// TwinCAT 3 PLC project CandyVendingMachine
// ProgramVersion: 3.1.4026.11
// libraries:
//   Tc2_Standard, * (Beckhoff Automation GmbH)
//   Tc2_System, * (Beckhoff Automation GmbH)
//   Tc2_Utilities, * (Beckhoff Automation GmbH)
// project tree:
//   AnyToArg/Classes/ AnyToTArgConverter.TcPOU
//   Candies/Classes/ AbstractCandy.TcPOU, Alpenliebe.TcPOU, Altoids.TcPOU, BobsSweetStripes.TcPOU, BrachsCandyCorn.TcPOU, ChupaChups.TcPOU, Goldbears.TcPOU, MnMs.TcPOU, Poppins.TcPOU, SkittlesSour.TcPOU, SnickersBar.TcPOU, TwizzlersLicorizeTwists.TcPOU, WonkaGobstopper.TcPOU
//   Candies/Types/Aliases/ CandyAmountInGram.TcDUT, CandyName.TcDUT
//   Candies/Types/Enums/ CandyTypes.TcDUT
//   CandyConsumer/Classes/ AbstractCandyConsumer.TcPOU
//   CandyConsumer/Types/Aliases/ ConsumerName.TcDUT, SatisfactionLevelInPercent.TcDUT
//   CandyDispatchers/Classes/ AbstractCandyDispatcher.TcPOU, CandyBarDispatcher.TcPOU, CandyCornDispatcher.TcPOU, CandyDispatcherFactory.TcPOU, CandySticksDispatcher.TcPOU, CaramelCandyDispatcher.TcPOU, ChoclateCandyDispatcher.TcPOU, GummyCandyDispatcher.TcPOU, HardCandyDispatcher.TcPOU, JawbreakersDispatcher.TcPOU, LicoriceCandyDispatcher.TcPOU, LollipopsDispatcher.TcPOU, MintsDispatcher.TcPOU, SourCandyDispatcher.TcPOU
//   CandyMachineProvider/Classes/ CandyMachineProvider.TcPOU, NinjaIncCandyMachineProvider.TcPOU
//   CandyMachine/Classes/ AbstractCandyMachine.TcPOU, CommonCandyMachine.TcPOU, GreedyCandyMachine.TcPOU, PickyCandyMachine.TcPOU
//   Logger/Classes/ AbstractLogger.TcPOU (not stored), AdsLogger.TcPOU, AdsLogMessage.TcPOU, LoggerProvider.TcPOU
//   NinjaCandyBehavior/Classes/ AbstractNinjaCandyConsumeBehavior.TcPOU, CommonNinjaCandyBehavior.TcPOU, GreedyNinjaCandyBehavior.TcPOU, PickyNinjaCandyBehavior.TcPOU
//   NinjaCandyBehavior/types/Enums/ ConsumerTypes.TcDUT, TasteScale.TcDUT
//   NinjaMonkeys/Classes/ AjninsCandyPreferences.TcPOU, IndividualCandyPreferences.TcPOU, NinjaMonkey.TcPOU
//   Tasks/Main/ MAIN.TcPOU, PlcTask.TcTTO
// real-time tasks:
//   TASK PlcTask: cycle T#10ms, priority 20, ADS port 350

CONFIGURATION CandyVendingMachine
    RESOURCE PLC ON TwinCAT3
        TASK PlcTask(INTERVAL := T#10ms, PRIORITY := 20);
        PROGRAM MAIN WITH PlcTask : MAIN;
    END_RESOURCE
END_CONFIGURATION

// ---- Candies/Types/Aliases/CandyAmountInGram.TcDUT
(*

short summary
=============
Alias of the subrange UINT(0..500).
It's used for the candy amount. The candy
machine is able to handle packaging units up
to 500 grams

legal notes
===========
SPDX-FileCopyrightText: © 2024 ekvip automation GmbH <info@ekvip.de>
SPDX-License-Identifier: Apache-2.0
For details check: Apache-2.0_

.. _Apache-2.0: https://www.apache.org/licenses/LICENSE-2.0

*)

TYPE CandyAmountInGram : 
	UINT(0..500); 
END_TYPE

// ---- Candies/Types/Aliases/CandyName.TcDUT
(*

short summary
=============
T_MaxString alias for the candy name.  

legal notes
===========
SPDX-FileCopyrightText: © 2024 ekvip automation GmbH <info@ekvip.de>
SPDX-License-Identifier: Apache-2.0
For details check: Apache-2.0_

.. _Apache-2.0: https://www.apache.org/licenses/LICENSE-2.0

*)

TYPE CandyName :
	Tc2_System.T_MaxString; 
END_TYPE

// ---- Candies/Types/Enums/CandyTypes.TcDUT
(*

short summary
=============
Enumeration of the candy types.
A single bit represents each candy type.
The candy type is stored in a word => so there can be
16 different candy types.
As a sweet usually consists of a mixture of different types, 
the enumeration is not strict. 
Each sweet can save its type by setting the corresponding bits. 

legal notes
===========
SPDX-FileCopyrightText: © 2024 ekvip automation GmbH <info@ekvip.de>
SPDX-License-Identifier: Apache-2.0
For details check: Apache-2.0_

.. _Apache-2.0: https://www.apache.org/licenses/LICENSE-2.0

*)

{attribute 'qualified_only'}
{attribute 'to_string'}
TYPE CandyTypes :
(
	(* bit 0 is type candy bar like a snickers *)
	CANDY_BARS		:= 16#0001,
	(* bit 1 is type candy corn like brach's candy corn *)
	CANDY_CORN		:= 16#0002,
	(* bit 2 is type stick candy like a christmas candy cane *)
	CANDY_STICKS	:= 16#0004,
	(* bit 3 is type caramel candy like omar cream *)
	CARAMEL_CANDY	:= 16#0008,
	(* bit 4 is type choclate candy like hershey *)
	CHOCOLATE_CANDY	:= 16#0010,
	(* bit 5 is type gummie candy like haribo *)
	GUMMY_CANDY		:= 16#0020,
	(* bit 6 is type mints like altoids *)
	MINTS			:= 16#0040,
	(* bit 7 is type lollipop like chupa chups *)
	LOLLIPOPS		:= 16#0080,
	(* bit 8 is type jawbreakers like willy wonka's everlasting gobstopper *) 
	JAWBREAKERS		:= 16#0100,
	(* bit 9 is type hard candy like pass pass pulse *)
	HARD_CANDY		:= 16#0200,
	(* bit 10 is type licorice candy like lakrids bülow *)
	LICORICE_CANDY	:= 16#0400,
	(* bit 11 is type sour candy like warheads *)
	SOUR_CANDY		:= 16#0800 	
)WORD;
END_TYPE

// ---- CandyConsumer/Types/Aliases/ConsumerName.TcDUT
(*

short summary
=============
A T_MaxString alias for the consumer name

legal notes
===========
SPDX-FileCopyrightText: © 2024 ekvip automation GmbH <info@ekvip.de>
SPDX-License-Identifier: Apache-2.0
For details check: Apache-2.0_

.. _Apache-2.0: https://www.apache.org/licenses/LICENSE-2.0

*)

TYPE ConsumerName :
	Tc2_System.T_MaxString; 
END_TYPE

// ---- CandyConsumer/Types/Aliases/SatisfactionLevelInPercent.TcDUT
(*

short summary
=============
alias for an unit subrange form 0 to 100.
It is used as satisfaction level for the candy consumer.
0 means depression
100 means euphoria

legal notes
===========
SPDX-FileCopyrightText: © 2024 ekvip automation GmbH <info@ekvip.de>
SPDX-License-Identifier: Apache-2.0
For details check: Apache-2.0_

.. _Apache-2.0: https://www.apache.org/licenses/LICENSE-2.0

*)

TYPE SatisfactionLevelInPercent :
	UINT(0..100); 
END_TYPE

// ---- NinjaCandyBehavior/types/Enums/ConsumerTypes.TcDUT
(*

short summary
=============
The world is full of different consumer types
but we've only defined two of it.
The greedy consumer (more is better)
The picky consumer (it's only worth it if it's good)

legal notes
===========
SPDX-FileCopyrightText: © 2024 ekvip automation GmbH <info@ekvip.de>
SPDX-License-Identifier: Apache-2.0
For details check: Apache-2.0_

.. _Apache-2.0: https://www.apache.org/licenses/LICENSE-2.0

*)

{attribute 'qualified_only'}
{attribute 'strict'}
{attribute 'to_string'}
TYPE ConsumerTypes :
(
	(* common neither picky nor greedy *)
	COMMON := 0,
	(* cookie monster style *)
	GREEDY,
	(* finicky style *)
	PICKY
)UDINT;
END_TYPE

// ---- NinjaCandyBehavior/types/Enums/TasteScale.TcDUT
(*

short summary
=============
This is enumeration is used as factor
to calculate the satisfaction level of the consumer.

legal notes
===========
SPDX-FileCopyrightText: © 2024 ekvip automation GmbH <info@ekvip.de>
SPDX-License-Identifier: Apache-2.0
For details check: Apache-2.0_

.. _Apache-2.0: https://www.apache.org/licenses/LICENSE-2.0

*)

{attribute 'qualified_only'}
{attribute 'strict'}
{attribute 'to_string'}
TYPE TasteScale :
(
	(* decreases maybe consumers statisfaction level *)
	DISGUSTING := -1,
	(* has maybe no effect on the consumers statisfaction level *)
	OKAY := 0,
	(* increases maybe consumers statisfaction level *)
	DELICIOUS := 1
)DINT := OKAY;
END_TYPE

// ---- Tasks/Main/MAIN.TcPOU
(*

short summary
=============
this is the main task of the
candy vending machine application

legal notes
===========
SPDX-FileCopyrightText: © 2024 ekvip automation GmbH <info@ekvip.de>
SPDX-License-Identifier: Apache-2.0
For details check: Apache-2.0_

.. _Apache-2.0: https://www.apache.org/licenses/LICENSE-2.0

*)

PROGRAM MAIN
VAR
	(* to print the log messages with the run method of the logger *)
	loggingProvider :LoggerProvider(0);
	(* behavior for a greedy candy consuming ninja *)
	greedy				:GreedyNinjaCandyBehavior(0);
	(* behavior for a picky candy consuming ninja *)
	picky				:PickyNinjaCandyBehavior(0);
	(* candy preferences of Ajnin *)
	ajninPreferences	:AjninsCandyPreferences();
	(* yeknom as candy consumer *)
	yeknom				:NinjaMonkey(greedy,0);
	(* ajnin as candy consumer *)
	ajnin				:NinjaMonkey(picky, ajninPreferences);
	(* rising edge will feed Ajnin *)
	feedAjnin			:BOOL;
	(* rising edge will feed Yeknom *)
	feedYeknom			:BOOL; 
END_VAR

ajnin.lootCandies(feedAjnin);
yeknom.lootCandies(feedYeknom);
loggingProvider.logger.run();

END_PROGRAM

// ---- Logger/Classes/LoggerProvider.TcPOU
(*

short summary
=============
A layer to hide the concrete used logger
and to make it easy to use the same logger

legal notes
===========
SPDX-FileCopyrightText: © 2024 ekvip automation GmbH <info@ekvip.de>
SPDX-License-Identifier: Apache-2.0
For details check: Apache-2.0_

.. _Apache-2.0: https://www.apache.org/licenses/LICENSE-2.0

*)

FUNCTION_BLOCK LoggerProvider
VAR_STAT
	(* differnt logger injected from outside *)
	injectedLogger	:REFERENCE TO AbstractLogger;
	(* default logger if nothing was injected *)
	defaultLogger 	:AdsLogger();
END_VAR

(*

short summary
=============
this method provides the possibility
to use a differnt logger for example
a file logger. 

legal notes
===========
SPDX-FileCopyrightText: © 2024 ekvip automation GmbH <info@ekvip.de>
SPDX-License-Identifier: Apache-2.0
For details check: Apache-2.0_

.. _Apache-2.0: https://www.apache.org/licenses/LICENSE-2.0

*)

METHOD FB_init :BOOL
VAR_INPUT
	(* if TRUE, the retain variables are initialized (warm start / cold start) *)
	bInitRetains	:BOOL;
	(* if TRUE, the instance afterwards gets moved into the copy code (online change) *) 
	bInCopyCode		:BOOL;
	(* if no other logger is required then use just 0 as parameter *)
	otherLogger		:REFERENCE TO AbstractLogger;
END_VAR
IF (__ISVALIDREF(otherLogger) AND_THEN NOT __ISVALIDREF(THIS^.injectedLogger)) THEN
	THIS^.injectedLogger REF= otherLogger;
END_IF
END_METHOD

(*

short summary
=============
property to get the used logger instance
 
legal notes
===========
SPDX-FileCopyrightText: © 2024 ekvip automation GmbH <info@ekvip.de>
SPDX-License-Identifier: Apache-2.0
For details check: Apache-2.0_

.. _Apache-2.0: https://www.apache.org/licenses/LICENSE-2.0

*)

PROPERTY logger :REFERENCE TO AbstractLogger
GET
(*

short summary
=============
getter of the property to get the used logger instance

legal notes
===========
SPDX-FileCopyrightText: © 2024 ekvip automation GmbH <info@ekvip.de>
SPDX-License-Identifier: Apache-2.0
For details check: Apache-2.0_

.. _Apache-2.0: https://www.apache.org/licenses/LICENSE-2.0

*)

VAR
END_VAR
IF (__ISVALIDREF(THIS^.injectedLogger)) THEN
	logger REF= THIS^.injectedLogger;
ELSE
	logger REF= THIS^.defaultLogger;
END_IF
END_GET
END_PROPERTY

END_FUNCTION_BLOCK

// ---- Logger/Classes/AdsLogger.TcPOU
(*

short summary
=============
a logger to write ADSLOG messages 

legal notes
===========
SPDX-FileCopyrightText: © 2024 ekvip automation GmbH <info@ekvip.de>
SPDX-License-Identifier: Apache-2.0
For details check: Apache-2.0_

.. _Apache-2.0: https://www.apache.org/licenses/LICENSE-2.0

*)

FUNCTION_BLOCK AdsLogger EXTENDS AbstractLogger
VAR
	(* buffer to store the messages *)
	messages		:POINTER TO POINTER TO AdsLogMessage;
	(* size of the message buffer *)
	size			:DWORD;
	(* the message buffer is a simple ring buffer this the read pointer for it *)
	readPointer		:DWORD := 0;
	(* the message buffer is a simple ring buffer this the write pointer for it *)
	writePointer	:DWORD := 0;
END_VAR
VAR CONSTANT
	(* inital message buffer size *) 
	MIN_BUFFER_SIZE :DWORD := 255;
END_VAR

(*

short summary
=============
this method appends a log message to the message buffer

legal notes
===========
SPDX-FileCopyrightText: © 2024 ekvip automation GmbH <info@ekvip.de>
SPDX-License-Identifier: Apache-2.0
For details check: Apache-2.0_

.. _Apache-2.0: https://www.apache.org/licenses/LICENSE-2.0

*)

METHOD PRIVATE appendNewMessage
VAR_INPUT
	(* ADSLOG message mask *)
	messageType :DWORD;
END_VAR
VAR_IN_OUT
	(* content of the log message *)
	message :Tc2_System.T_MaxString;
END_VAR
VAR
	(* pointer to the new log message *) 
	new	:POINTER TO AdsLogMessage;
END_VAR
IF (THIS^.isBufferFull OR (THIS^.messages = 0)) THEN
	THIS^.resize();
END_IF
RETURN((THIS^.messages = 0) OR_ELSE THIS^.isBufferFull);

new := __NEW(AdsLogMessage(msg := message, msgType := messageType));
RETURN(new = 0);
THIS^.messages[THIS^.writePointer] := new;
THIS^.writePointer := THIS^.incrementBufferPointer(THIS^.writePointer);
END_METHOD

(*

short summary
=============
writes a log message for a critical event
It will be stored in the twinCAT logbook 
and open a message box

legal notes
===========
SPDX-FileCopyrightText: © 2024 ekvip automation GmbH <info@ekvip.de>
SPDX-License-Identifier: Apache-2.0
For details check: Apache-2.0_

.. _Apache-2.0: https://www.apache.org/licenses/LICENSE-2.0

*)

METHOD critical
VAR_INPUT
	(* log message to write *)
	message :Tc2_System.T_MaxString;
END_VAR
THIS^.appendNewMessage(
	Tc2_System.ADSLOG_MSGTYPE_ERROR OR Tc2_System.ADSLOG_MSGTYPE_RESOURCE OR Tc2_System.ADSLOG_MSGTYPE_MSGBOX, 
	message
);
END_METHOD

(*

short summary
=============
method to log a debug message

legal notes
===========
SPDX-FileCopyrightText: © 2024 ekvip automation GmbH <info@ekvip.de>
SPDX-License-Identifier: Apache-2.0
For details check: Apache-2.0_

.. _Apache-2.0: https://www.apache.org/licenses/LICENSE-2.0

*)

METHOD debug
VAR_INPUT
	(* log message to write *)
	message :Tc2_System.T_MaxString;
END_VAR
THIS^.appendNewMessage(Tc2_System.ADSLOG_MSGTYPE_HINT, message);
END_METHOD

(*

short summary
=============
method to log a error message

legal notes
===========
SPDX-FileCopyrightText: © 2024 ekvip automation GmbH <info@ekvip.de>
SPDX-License-Identifier: Apache-2.0
For details check: Apache-2.0_

.. _Apache-2.0: https://www.apache.org/licenses/LICENSE-2.0

*)

METHOD error
VAR_INPUT
	(* log message to write *)
	message :Tc2_System.T_MaxString;
END_VAR
THIS^.appendNewMessage(Tc2_System.ADSLOG_MSGTYPE_ERROR, message);
END_METHOD

(*

short summary
=============
this method clean up the memory
(free it again)

legal notes
===========
SPDX-FileCopyrightText: © 2024 ekvip automation GmbH <info@ekvip.de>
SPDX-License-Identifier: Apache-2.0
For details check: Apache-2.0_

.. _Apache-2.0: https://www.apache.org/licenses/LICENSE-2.0

*)

METHOD FB_exit :BOOL
VAR_INPUT
	(* if TRUE, the exit method is called for exiting an instance that is copied afterwards (online change). *)
	bInCopyCode :BOOL;
END_VAR
VAR
	(* buffer pointer to free the message buffer memory again *)
	buffer 		:POINTER TO __XWORD;
END_VAR
RETURN(THIS^.messages = 0);
WHILE (NOT THIS^.isBufferEmpty) DO
	THIS^.printMessage();
END_WHILE
buffer := THIS^.messages;
__DELETE(buffer);
THIS^.messages := 0;
THIS^.size := 0;
THIS^.writePointer := 0;
THIS^.readPointer := 0;
END_METHOD

(*

short summary
=============
method to increment the read and write pointer
of the message buffer

legal notes
===========
SPDX-FileCopyrightText: © 2024 ekvip automation GmbH <info@ekvip.de>
SPDX-License-Identifier: Apache-2.0
For details check: Apache-2.0_

.. _Apache-2.0: https://www.apache.org/licenses/LICENSE-2.0

*)

METHOD PRIVATE incrementBufferPointer :DWORD
VAR_INPUT
	(* current pointer value *)
	bufferPointer :DWORD;
END_VAR
incrementBufferPointer := ((bufferPointer + 1) MOD THIS^.size);
END_METHOD

(*

short summary
=============
method to log a info message

legal notes
===========
SPDX-FileCopyrightText: © 2024 ekvip automation GmbH <info@ekvip.de>
SPDX-License-Identifier: Apache-2.0
For details check: Apache-2.0_

.. _Apache-2.0: https://www.apache.org/licenses/LICENSE-2.0

*)

METHOD info
VAR_INPUT
	(* log message to write *)
	message :Tc2_System.T_MaxString;
END_VAR
THIS^.appendNewMessage(Tc2_System.ADSLOG_MSGTYPE_HINT, message);
END_METHOD

(*

short summary
=============
property to check if the
ring buffer is empty

legal notes
===========
SPDX-FileCopyrightText: © 2024 ekvip automation GmbH <info@ekvip.de>
SPDX-License-Identifier: Apache-2.0
For details check: Apache-2.0_

.. _Apache-2.0: https://www.apache.org/licenses/LICENSE-2.0

*)

PROPERTY PRIVATE isBufferEmpty :BOOL
GET
(*

short summary
=============
getter of the property to check if the
ring buffer is empty

legal notes
===========
SPDX-FileCopyrightText: © 2024 ekvip automation GmbH <info@ekvip.de>
SPDX-License-Identifier: Apache-2.0
For details check: Apache-2.0_

.. _Apache-2.0: https://www.apache.org/licenses/LICENSE-2.0

*)

VAR
END_VAR
isBufferEmpty := (THIS^.readPointer = THIS^.writePointer);
END_GET
END_PROPERTY

(*

short summary
=============
property to check if the
ring buffer is full

legal notes
===========
SPDX-FileCopyrightText: © 2024 ekvip automation GmbH <info@ekvip.de>
SPDX-License-Identifier: Apache-2.0
For details check: Apache-2.0_

.. _Apache-2.0: https://www.apache.org/licenses/LICENSE-2.0

*)

PROPERTY PRIVATE isBufferFull :BOOL
GET
(*

short summary
=============
getter of the property to check if the
ring buffer is full

legal notes
===========
SPDX-FileCopyrightText: © 2024 ekvip automation GmbH <info@ekvip.de>
SPDX-License-Identifier: Apache-2.0
For details check: Apache-2.0_

.. _Apache-2.0: https://www.apache.org/licenses/LICENSE-2.0

*)

VAR
END_VAR
isBufferFull := (THIS^.incrementBufferPointer(THIS^.writePointer) = THIS^.readPointer);
END_GET
END_PROPERTY

(*

short summary
=============
method to write the log message to
ADSLOG and it frees the memory of
the message again

legal notes
===========
SPDX-FileCopyrightText: © 2024 ekvip automation GmbH <info@ekvip.de>
SPDX-License-Identifier: Apache-2.0
For details check: Apache-2.0_

.. _Apache-2.0: https://www.apache.org/licenses/LICENSE-2.0

*)

METHOD PRIVATE printMessage
VAR
	(* message pointer to free the memory again *)
	msg :POINTER TO AdsLogMessage;
END_VAR
IF (THIS^.messages[THIS^.readPointer] <> 0) THEN
	Tc2_System.ADSLOGSTR(
		msgCtrlMask := THIS^.messages[THIS^.readPointer]^.messageType,
		msgFmtStr := '%s',
		strArg := THIS^.messages[THIS^.readPointer]^.message
	);
	msg := THIS^.messages[THIS^.readPointer];
	__DELETE(msg);
	THIS^.messages[THIS^.readPointer] := 0;
END_IF
THIS^.readPointer := THIS^.incrementBufferPointer(THIS^.readPointer);
END_METHOD

(*

short summary
=============
this method resizes the messages buffer
if it is full or not created

legal notes
===========
SPDX-FileCopyrightText: © 2024 ekvip automation GmbH <info@ekvip.de>
SPDX-License-Identifier: Apache-2.0
For details check: Apache-2.0_

.. _Apache-2.0: https://www.apache.org/licenses/LICENSE-2.0

*)

METHOD PRIVATE resize
VAR
	(* new buffer for the messages array *)
	newBuffer 			:POINTER TO __XWORD;
	(* just to free the memory again *)
	oldBuffer 			:POINTER TO __XWORD;
	(* pointer with the smaller value *)
	minPointer  		:DWORD;
	(* pointer with the bigger value *)
	maxPointer  		:DWORD;
	(* new position in new message buffer of the pointer with the bigger value *)
	newMaxPointerPos	:DWORD;
	(* number of elements to copy for the pointer with the bigger value *)
	amountMaxPointer	:DWORD;
	(* new size of the messages buffer *)
	newSize 			:DWORD;
END_VAR
newSize := MAX(THIS^.MIN_BUFFER_SIZE, THIS^.size * 2);
RETURN(newSize < THIS^.size);
newBuffer := __NEW(__XWORD, newSize);
RETURN(newBuffer = 0);
IF (NOT THIS^.isBufferEmpty) THEN
	minPointer := MIN(THIS^.writePointer, THIS^.readPointer);
	maxPointer := MAX(THIS^.writePointer, THIS^.readPointer);
	amountMaxPointer := SEL(
		((THIS^.size-1) = maxPointer),
		((THIS^.size-1)-maxPointer),
		THIS^.size-1
	);
	newMaxPointerPos := ((newSize-1)-amountMaxPointer);
	Tc2_System.MEMCPY(
		destAddr	:= newBuffer,
		srcAddr		:= THIS^.messages,
		n			:= ((minPointer+1)*SIZEOF(__XWORD))
	);
	Tc2_System.MEMCPY(
		destAddr	:= ADR(newBuffer[SEL(((THIS^.size-1) = maxPointer),newMaxPointerPos,minPointer+1)]),
		srcAddr		:= ADR(THIS^.messages[minPointer+1]),
		n			:= (amountMaxPointer*SIZEOF(__XWORD))
	);
	IF (THIS^.readPointer > THIS^.writePointer) THEN
		THIS^.readPointer := newMaxPointerPos;
	ELSE
		THIS^.writePointer := newMaxPointerPos;
	END_IF
END_IF
IF (THIS^.messages <> 0) THEN
	oldBuffer := THIS^.messages;
	__DELETE(oldBuffer);
END_IF
THIS^.messages := newBuffer;
THIS^.size := newSize;
END_METHOD

(*

short summary
=============
fetches the messages from buffer and
writes it to ADSLOG. This method must
be called cyclic.

legal notes
===========
SPDX-FileCopyrightText: © 2024 ekvip automation GmbH <info@ekvip.de>
SPDX-License-Identifier: Apache-2.0
For details check: Apache-2.0_

.. _Apache-2.0: https://www.apache.org/licenses/LICENSE-2.0

*)

METHOD run
VAR_INST
	(* TON timer to write the messages in a serial way *)
	printNextMsg	:Tc2_Standard.TON;	
END_VAR
RETURN(THIS^.messages = 0);
printNextMsg(IN:= TRUE, PT:=T#30MS);
RETURN(NOT printNextMsg.Q);
RETURN(THIS^.isBufferEmpty);
printNextMsg(IN:= FALSE);
THIS^.printMessage();
END_METHOD

(*

short summary
=============
method to log a warning message

legal notes
===========
SPDX-FileCopyrightText: © 2024 ekvip automation GmbH <info@ekvip.de>
SPDX-License-Identifier: Apache-2.0
For details check: Apache-2.0_

.. _Apache-2.0: https://www.apache.org/licenses/LICENSE-2.0

*)

METHOD warning
VAR_INPUT
	(* log message to write *)
	message :Tc2_System.T_MaxString;
END_VAR
THIS^.appendNewMessage(Tc2_System.ADSLOG_MSGTYPE_WARN, message);
END_METHOD

END_FUNCTION_BLOCK

// ---- Logger/Classes/AdsLogMessage.TcPOU
(*

short summary
=============
just a dto to store the logging data for
the ads logger

legal notes
===========
SPDX-FileCopyrightText: © 2024 ekvip automation GmbH <info@ekvip.de>
SPDX-License-Identifier: Apache-2.0
For details check: Apache-2.0_

.. _Apache-2.0: https://www.apache.org/licenses/LICENSE-2.0

*)

{attribute 'enable_dynamic_creation'}
FUNCTION_BLOCK AdsLogMessage
VAR
	(* log message content *)
	msg		:Tc2_System.T_MaxString;
	(* ADSLOG message type mask *)
	msgType	:DWORD;
END_VAR

(*

short summary
=============
initialize the message values

legal notes
===========
SPDX-FileCopyrightText: © 2024 ekvip automation GmbH <info@ekvip.de>
SPDX-License-Identifier: Apache-2.0
For details check: Apache-2.0_

.. _Apache-2.0: https://www.apache.org/licenses/LICENSE-2.0

*)

METHOD FB_init :BOOL
VAR_INPUT
	(* if TRUE, the retain variables are initialized (warm start / cold start) *)
	bInitRetains	:BOOL;
	(* if TRUE, the instance afterwards gets moved into the copy code (online change) *) 
	bInCopyCode		:BOOL;
	(* content of the message *)
	msg				:Tc2_System.T_MaxString;
	(* mask of an ADSLOG *)
	msgType			:DWORD;
END_VAR
THIS^.msg := msg;
THIS^.msgType := msgType;
END_METHOD

(*

short summary
=============
property to get the message content

legal notes
===========
SPDX-FileCopyrightText: © 2024 ekvip automation GmbH <info@ekvip.de>
SPDX-License-Identifier: Apache-2.0
For details check: Apache-2.0_

.. _Apache-2.0: https://www.apache.org/licenses/LICENSE-2.0

*)

PROPERTY message :Tc2_System.T_MaxString
GET
(*

short summary
=============
getter of the property to get the message content

legal notes
===========
SPDX-FileCopyrightText: © 2024 ekvip automation GmbH <info@ekvip.de>
SPDX-License-Identifier: Apache-2.0
For details check: Apache-2.0_

.. _Apache-2.0: https://www.apache.org/licenses/LICENSE-2.0

*)

VAR
END_VAR
message := THIS^.msg;
END_GET
END_PROPERTY

(*

short summary
=============
property to get the ads message type mask

legal notes
===========
SPDX-FileCopyrightText: © 2024 ekvip automation GmbH <info@ekvip.de>
SPDX-License-Identifier: Apache-2.0
For details check: Apache-2.0_

.. _Apache-2.0: https://www.apache.org/licenses/LICENSE-2.0

*)

PROPERTY messageType :DWORD
GET
(*

short summary
=============
getter of the property to get the ads message type mask

legal notes
===========
SPDX-FileCopyrightText: © 2024 ekvip automation GmbH <info@ekvip.de>
SPDX-License-Identifier: Apache-2.0
For details check: Apache-2.0_

.. _Apache-2.0: https://www.apache.org/licenses/LICENSE-2.0

*)

VAR
END_VAR
messageType := THIS^.msgType;
END_GET
END_PROPERTY

END_FUNCTION_BLOCK

// ---- NinjaCandyBehavior/Classes/GreedyNinjaCandyBehavior.TcPOU
(*

short summary
=============
the behavior of a greedy ninja

legal notes
===========
SPDX-FileCopyrightText: © 2024 ekvip automation GmbH <info@ekvip.de>
SPDX-License-Identifier: Apache-2.0
For details check: Apache-2.0_

.. _Apache-2.0: https://www.apache.org/licenses/LICENSE-2.0

*)

FUNCTION_BLOCK GreedyNinjaCandyBehavior EXTENDS AbstractNinjaCandyConsumeBehavior
VAR_STAT
	(* default provider for the greedies*)
	greedyDefaultProvider :NinjaIncCandyMachineProvider(ConsumerTypes.GREEDY);
END_VAR

(*

short summary
=============
This method calculates the satisfaction level
for a candy eating greedy consumer.

legal notes
===========
SPDX-FileCopyrightText: © 2024 ekvip automation GmbH <info@ekvip.de>
SPDX-License-Identifier: Apache-2.0
For details check: Apache-2.0_

.. _Apache-2.0: https://www.apache.org/licenses/LICENSE-2.0

*)

METHOD  calculateSatisfactionLevel
VAR_INPUT
	(* taste scale of candy *)
	tastiness				:TasteScale;
	(* amount of the candies to eat *)
	amountOfCandy			:CandyAmountInGram;
END_VAR
VAR_IN_OUT
	(* the satisfaction level of the consumer *)
	actualSatisfactionLevel	:SatisfactionLevelInPercent;
END_VAR
VAR CONSTANT
	(* maximum possible satisfaction level*)
	MAX_SATISFACTION 		:SatisfactionLevelInPercent := 100;
	(* it is a lower limit as it is named *)
	AVOID_DIVISON_BY_ZERO 	:SatisfactionLevelInPercent := 1;
	(* factor for the greediness of the consumer *)
	GREEDINESS				:SatisfactionLevelInPercent := 78;
	(* for one a candy package the maximum amount *)
	MAX_AMOUNT				:CandyAmountInGram := 500;
END_VAR
RETURN(actualSatisfactionLevel >= MAX_SATISFACTION);

{warning disable C0196}
{warning disable C0197}
actualSatisfactionLevel := TO_UINT(
	actualSatisfactionLevel + TO_SINT(
		LOG(
			TO_REAL(MAX_SATISFACTION)
			/TO_REAL(LIMIT(AVOID_DIVISON_BY_ZERO, actualSatisfactionLevel, MAX_SATISFACTION))
		) * (
			TO_REAL(amountOfCandy)
			/TO_REAL(MAX_AMOUNT)
		)
		* (MAX_SATISFACTION - GREEDINESS)
	)
);
{warning restore C0196}
{warning restore C0197}
END_METHOD

(*

short summary
=============
inject the candy vending machine provider
during declaration.

legal notes
===========
SPDX-FileCopyrightText: © 2024 ekvip automation GmbH <info@ekvip.de>
SPDX-License-Identifier: Apache-2.0
For details check: Apache-2.0_

.. _Apache-2.0: https://www.apache.org/licenses/LICENSE-2.0

*)

METHOD FB_init :BOOL
VAR_INPUT
	(* if TRUE, the retain variables are initialized (warm start / cold start) *)
	bInitRetains		:BOOL;
	(* if TRUE, the instance afterwards gets moved into the copy code (online change) *)
	bInCopyCode			:BOOL;
	(* candy vending machine provider for the consumer *)
	candyMachineProvider:REFERENCE TO CandyMachineProvider;
END_VAR
IF (__ISVALIDREF(candyMachineProvider)) THEN
	THIS^.candyMachineProvider REF= candyMachineProvider;
ELSE
	THIS^.candyMachineProvider REF= THIS^.greedyDefaultProvider;
END_IF
END_METHOD

END_FUNCTION_BLOCK

// ---- NinjaCandyBehavior/Classes/AbstractNinjaCandyConsumeBehavior.TcPOU
(*

short summary
=============
different consumers have a different
behavior. This class is to decouple
behavior from the consumer.

legal notes
===========
SPDX-FileCopyrightText: © 2024 ekvip automation GmbH <info@ekvip.de>
SPDX-License-Identifier: Apache-2.0
For details check: Apache-2.0_

.. _Apache-2.0: https://www.apache.org/licenses/LICENSE-2.0

*)

FUNCTION_BLOCK ABSTRACT AbstractNinjaCandyConsumeBehavior
VAR
	(* candy vending machine provider to get a machine to loot *)
	candyMachineProvider	:REFERENCE TO CandyMachineProvider;
END_VAR
VAR_STAT
	(* default provider *)
	defaultProvider :NinjaIncCandyMachineProvider(ConsumerTypes.COMMON);
END_VAR

(*

short summary
=============
This method calculates the satisfaction level if the consumer
eates some candies.

legal notes
===========
SPDX-FileCopyrightText: © 2024 ekvip automation GmbH <info@ekvip.de>
SPDX-License-Identifier: Apache-2.0
For details check: Apache-2.0_

.. _Apache-2.0: https://www.apache.org/licenses/LICENSE-2.0

*)

METHOD ABSTRACT calculateSatisfactionLevel
VAR_INPUT
	(* taste scale of candy *)
	tastiness				:TasteScale;
	(* amount of the candies to eat *)
	amountOfCandy			:CandyAmountInGram;
END_VAR
VAR_IN_OUT
	(* the satisfaction level of the consumer *)
	actualSatisfactionLevel	:SatisfactionLevelInPercent;
END_VAR
END_METHOD

(*

short summary
=============
inject the candy vending machine provider
during declaration.

legal notes
===========
SPDX-FileCopyrightText: © 2024 ekvip automation GmbH <info@ekvip.de>
SPDX-License-Identifier: Apache-2.0
For details check: Apache-2.0_

.. _Apache-2.0: https://www.apache.org/licenses/LICENSE-2.0

*)

METHOD FB_init :BOOL
VAR_INPUT
	(* if TRUE, the retain variables are initialized (warm start / cold start) *)
	bInitRetains		:BOOL;
	(* if TRUE, the instance afterwards gets moved into the copy code (online change) *)
	bInCopyCode			:BOOL;
	(* candy vending machine provider for the consumer *)
	candyMachineProvider:REFERENCE TO CandyMachineProvider;
END_VAR
IF (__ISVALIDREF(candyMachineProvider)) THEN
	THIS^.candyMachineProvider REF= candyMachineProvider;
ELSE
	THIS^.candyMachineProvider REF= THIS^.defaultProvider;
END_IF
END_METHOD

(*

short summary
=============
this method is for the looting behavior
of the picky consumer. 
The picky consumer tries to by delcious candy only.

legal notes
===========
SPDX-FileCopyrightText: © 2024 ekvip automation GmbH <info@ekvip.de>
SPDX-License-Identifier: Apache-2.0
For details check: Apache-2.0_

.. _Apache-2.0: https://www.apache.org/licenses/LICENSE-2.0

*)

METHOD  lootACandyMachine
VAR_INPUT
	(* consumer who loots a candy vending machine *)
	consumer :REFERENCE TO AbstractCandyConsumer;
	(* preferences of consumer no preference means consumer likes every candy *)
	preferences	:REFERENCE TO IndividualCandyPreferences REF= 0;
END_VAR
VAR
	(* for-loop counter *)
	candyToEat		:CandyTypes;
	(* used candy vending machine *)
	candyMachine	:REFERENCE TO AbstractCandyMachine;
	(* the candy to eat *)
	candy			:REFERENCE TO AbstractCandy;
END_VAR
RETURN(NOT __ISVALIDREF(consumer));
candyMachine REF= THIS^.candyMachineProvider.getACandyMachine();
RETURN(NOT __ISVALIDREF(candyMachine));

FOR candyToEat := CandyTypes.CANDY_BARS TO CandyTypes.SOUR_CANDY BY candyToEat DO
	IF (__ISVALIDREF(preferences) AND_THEN preferences.howIsTheCandy(candyToEat) <> TasteScale.DELICIOUS) THEN
		CONTINUE;
	END_IF
	candy REF= candyMachine.getNewCandy(candyToEat);
	IF (__ISVALIDREF(candy)) THEN
		candy.eatMe(consumer);
	END_IF
END_FOR
END_METHOD

END_FUNCTION_BLOCK

// ---- CandyMachineProvider/Classes/CandyMachineProvider.TcPOU
(*

short summary
=============
the candy machine provider provides
candy vending machines for different candy 
consumers (greedy or picky eaters)

legal notes
===========
SPDX-FileCopyrightText: © 2024 ekvip automation GmbH <info@ekvip.de>
SPDX-License-Identifier: Apache-2.0
For details check: Apache-2.0_

.. _Apache-2.0: https://www.apache.org/licenses/LICENSE-2.0

*)

FUNCTION_BLOCK ABSTRACT CandyMachineProvider
VAR
	(* this for the case that a special candy machine for special consumers is required *)
	{attribute 'hide'}
	customCandyMachine	:REFERENCE TO AbstractCandyMachine REF= 0;
END_VAR
VAR_STAT
	(* this is the candy machine for every body *)
	{attribute 'hide'}
	defaultCandyMachine :CommonCandyMachine();
END_VAR

(*

short summary
=============
this method provides returns a candy vending machine

legal notes
===========
SPDX-FileCopyrightText: © 2024 ekvip automation GmbH <info@ekvip.de>
SPDX-License-Identifier: Apache-2.0
For details check: Apache-2.0_

.. _Apache-2.0: https://www.apache.org/licenses/LICENSE-2.0

*)

METHOD getACandyMachine :REFERENCE TO AbstractCandyMachine
IF (__ISVALIDREF(THIS^.customCandyMachine)) THEN
	getACandyMachine REF= THIS^.customCandyMachine;
ELSE
	getACandyMachine REF= THIS^.defaultCandyMachine;
END_IF
END_METHOD

END_FUNCTION_BLOCK

// ---- CandyMachine/Classes/AbstractCandyMachine.TcPOU
(*

short summary
=============
candy vending machine it provides
candies for every taste

legal notes
===========
SPDX-FileCopyrightText: © 2024 ekvip automation GmbH <info@ekvip.de>
SPDX-License-Identifier: Apache-2.0
For details check: Apache-2.0_

.. _Apache-2.0: https://www.apache.org/licenses/LICENSE-2.0

*)

FUNCTION_BLOCK ABSTRACT AbstractCandyMachine

(*

short summary
=============
this method provides candies.
Just select your preferred pure candy type

legal notes
===========
SPDX-FileCopyrightText: © 2024 ekvip automation GmbH <info@ekvip.de>
SPDX-License-Identifier: Apache-2.0
For details check: Apache-2.0_

.. _Apache-2.0: https://www.apache.org/licenses/LICENSE-2.0

*)

METHOD ABSTRACT getNewCandy :REFERENCE TO AbstractCandy
VAR_INPUT
	(*preferred candy type, it must be a pure candy type *)
	candyType	:CandyTypes;
END_VAR
END_METHOD

(*

short summary
=============
helper method to test if the candy type 
value is in the range and is a power of 2.
- it returns true if the value is invalid
- it returns false if value is valid

legal notes
===========
SPDX-FileCopyrightText: © 2024 ekvip automation GmbH <info@ekvip.de>
SPDX-License-Identifier: Apache-2.0
For details check: Apache-2.0_

.. _Apache-2.0: https://www.apache.org/licenses/LICENSE-2.0

*)

METHOD PROTECTED isCandyTypeInvalidForMachine :BOOL
VAR_INPUT
	(* candy type value to test *)
	candyType	:CandyTypes;
END_VAR
isCandyTypeInvalidForMachine := TRUE;
RETURN((candyType < CandyTypes.CANDY_BARS) OR (candyType > CandyTypes.SOUR_CANDY));
RETURN((candyType AND (candyType-1)) <> 0);
isCandyTypeInvalidForMachine := FALSE;
END_METHOD

END_FUNCTION_BLOCK

// ---- Candies/Classes/AbstractCandy.TcPOU
(*

short summary
=============
This class is an abstraction layer for candies.
Every candy must inherit from it.
Every candy must have the attribute pragma call after init
because it's impossible to create the dispatchers in FB_init.
If a concrete candy was created dynamically then it's necessary
to call the method initializeDispatchers once. 

legal notes
===========
SPDX-FileCopyrightText: © 2024 ekvip automation GmbH <info@ekvip.de>
SPDX-License-Identifier: Apache-2.0
For details check: Apache-2.0_

.. _Apache-2.0: https://www.apache.org/licenses/LICENSE-2.0

*)
{attribute 'call_after_init'}
FUNCTION_BLOCK ABSTRACT AbstractCandy EXTENDS AnyToTArgConverter
VAR
	(* common candy type for example caramel candy *)
	candyType		:CandyTypes;
	(* name of the candy like snickers *)
	name			:CandyName;
	(* amount of the candy in gram because we use the metric system *)
	amount			:CandyAmountInGram;
	(* array of dispatchers to dispatch a common candy type to a consumer *)
	{attribute 'no_copy'}
	dispatcher		:POINTER TO POINTER TO AbstractCandyDispatcher;
	(* factory to create the dispatchers dynamically *)
	{attribute 'hide'}
	dispatcherFactory :CandyDispatcherFactory();
	(*
	number common candy types of the concrete candy.
	For example a snickers is a candy bar, a chocolate candy and a caramel candy, 
	in this example the numberOfTypes is three
	*)
	numberOfTypes	:USINT;
END_VAR

(*

short summary
=============
This method adds a dispatcher for a specific candy type
to the the concrete candy. It's possible that a concrete
candy has more than one specific candy type. For example a 
snickers is a candy bar, a caramel candy and chocolate candy.
Since the consumer has for every candy type a extra method
to call, the class AbtractCandy use dispatchers classes
to simplify it. The dispatcher is a pointer to pointer to
make it iterable because it's impossible do it with an
array of references to AbstractCandyDispatcher.

legal notes
===========
SPDX-FileCopyrightText: © 2024 ekvip automation GmbH <info@ekvip.de>
SPDX-License-Identifier: Apache-2.0
For details check: Apache-2.0_

.. _Apache-2.0: https://www.apache.org/licenses/LICENSE-2.0

*)
METHOD PRIVATE addNewDispatcher
VAR_INPUT
	(* candy type to add a new dispatcher for it *)
	candyType	:CandyTypes;
END_VAR
VAR
	(* pointer to an abstract dispatcher to store it in the array (pointer to pointer) *)
	dispatcher	:POINTER TO AbstractCandyDispatcher;
	(* array for the abstract dispatchers *)
	dispatchers	:POINTER TO __XWORD;
END_VAR
dispatcher := THIS^.dispatcherFactory.getNewCandyDispatcherFor(candyType);
RETURN (dispatcher <= 0);
dispatchers := __NEW(__XWORD, (THIS^.numberOfTypes + 1));
IF (THIS^.dispatcher > 0) THEN
	Tc2_System.MEMCPY(
		destAddr := dispatchers,
		srcAddr := THIS^.dispatcher,
		n := (SIZEOF(__XWORD)*THIS^.numberOfTypes)
	);
	__DELETE(THIS^.dispatcher);
END_IF
dispatchers[THIS^.numberOfTypes] := dispatcher;
THIS^.numberOfTypes := (THIS^.numberOfTypes + 1);
THIS^.dispatcher := dispatchers;
END_METHOD

(*

short summary
=============
This property has just a getter, and it returns the
amount of the candy in gram. For example a package
Alpenliebe Gold contains 156 gram, so a instance of
a Alpenliebe class will return 156.

legal notes
===========
SPDX-FileCopyrightText: © 2024 ekvip automation GmbH <info@ekvip.de>
SPDX-License-Identifier: Apache-2.0
For details check: Apache-2.0_

.. _Apache-2.0: https://www.apache.org/licenses/LICENSE-2.0

*)
PROPERTY amountOfCandy : CandyAmountInGram
GET
(*

short summary
=============
The getter for the candy amount.

legal notes
===========
SPDX-FileCopyrightText: © 2024 ekvip automation GmbH <info@ekvip.de>
SPDX-License-Identifier: Apache-2.0
For details check: Apache-2.0_

.. _Apache-2.0: https://www.apache.org/licenses/LICENSE-2.0

*)
VAR
END_VAR
amountOfCandy := THIS^.amount;
END_GET
END_PROPERTY

(*

short summary
=============
This method is to free the memory of an abstract candy again
if the candy was dynamically created. The method has no effect
if the candy was not dynamically created. It returns a null pointer
if it free the memory and a pointer to it self if it didn't free
memory. The method simplify the destruction of a candy object
because it is no query pointer neccessary.

legal notes
===========
SPDX-FileCopyrightText: © 2024 ekvip automation GmbH <info@ekvip.de>
SPDX-License-Identifier: Apache-2.0
For details check: Apache-2.0_

.. _Apache-2.0: https://www.apache.org/licenses/LICENSE-2.0

*)
METHOD PROTECTED destruct :POINTER TO AbstractCandy
VAR CONSTANT
	(* value of a null pointer *)
	NULL :__XWORD := 0;
END_VAR
destruct := THIS;
IF (
	Tc2_System.F_CheckMemoryArea(pData := THIS, nSize := SIZEOF(THIS^))
	= Tc2_System.E_TcMemoryArea.Dynamic
) THEN
	__DELETE(destruct);
	destruct := NULL;
END_IF
END_METHOD

(*

short summary
=============
this method calls the eat<CandyType> methods of
the candy consumer and it destruct the candy object.

legal notes
===========
SPDX-FileCopyrightText: © 2024 ekvip automation GmbH <info@ekvip.de>
SPDX-License-Identifier: Apache-2.0
For details check: Apache-2.0_

.. _Apache-2.0: https://www.apache.org/licenses/LICENSE-2.0

*)

METHOD eatMe :POINTER TO AbstractCandy
VAR_INPUT
	(* candy consumer who eats the candy *)
	consumer :REFERENCE TO AbstractCandyConsumer;
END_VAR
VAR
	i	:USINT;
END_VAR
eatMe := THIS;
RETURN(NOT __ISVALIDREF(consumer));
RETURN(THIS^.numberOfTypes <= 0);

FOR i:= 0 TO (THIS^.numberOfTypes-1) DO
	THIS^.dispatcher[i]^.eat(consumer, (THIS^.amount / THIS^.numberOfTypes));
END_FOR

THIS^.logCandyConsume(consumer);
eatMe := THIS^.destruct();
END_METHOD

(*

short summary
=============
frees the memory of the candy dispatcher again.

legal notes
===========
SPDX-FileCopyrightText: © 2024 ekvip automation GmbH <info@ekvip.de>
SPDX-License-Identifier: Apache-2.0
For details check: Apache-2.0_

.. _Apache-2.0: https://www.apache.org/licenses/LICENSE-2.0

*)

METHOD FB_exit : BOOL
VAR_INPUT
	(* if TRUE, the exit method is called for exiting an instance that is copied afterwards (online change). *)
	bInCopyCode : BOOL;
END_VAR
THIS^.freeDispatchers();
END_METHOD

(*

short summary
=============
destruc the dynamicly created dispatcher to
free the memory again.

legal notes
===========
SPDX-FileCopyrightText: © 2024 ekvip automation GmbH <info@ekvip.de>
SPDX-License-Identifier: Apache-2.0
For details check: Apache-2.0_

.. _Apache-2.0: https://www.apache.org/licenses/LICENSE-2.0

*)

METHOD PRIVATE freeDispatchers
VAR_INPUT
END_VAR
VAR
	(* counter vairable for the for-loop *)
	currentDispatcher :USINT;
	(* memory was allocated as __XWORD so a __XWORD pointer is required to free it again *)
	dispatchers	:POINTER TO __XWORD;
END_VAR
RETURN(THIS^.numberOfTypes <= 0);
RETURN(THIS^.dispatcher <= 0);
FOR currentDispatcher := 0 TO THIS^.numberOfTypes-1 DO
	THIS^.dispatcher[currentDispatcher]^.destruct();
END_FOR
THIS^.numberOfTypes := 0;
dispatchers := THIS^.dispatcher;
__DELETE(dispatchers);
THIS^.dispatcher := 0;
END_METHOD

(*

short summary
=============
creates the dispatcher dynamicly for the candy.
It is not possible to do this in FB_init because
of the order (base class first)

legal notes
===========
SPDX-FileCopyrightText: © 2024 ekvip automation GmbH <info@ekvip.de>
SPDX-License-Identifier: Apache-2.0
For details check: Apache-2.0_

.. _Apache-2.0: https://www.apache.org/licenses/LICENSE-2.0

*)

{attribute 'call_after_init'}
METHOD initializeDispatchers
VAR_INPUT
END_VAR
VAR
	(* counter variable for binary counting in a for-loop *)
	currentType	:CandyTypes;
	(* binary candy types from FB_init *)
	myCandyType :CandyTypes := THIS^.candyType;
END_VAR
THIS^.freeDispatchers();
RETURN(myCandyType <= 0);
FOR currentType := CandyTypes.CANDY_BARS TO CandyTypes.SOUR_CANDY BY currentType DO
	IF ((myCandyType AND currentType) > 0) THEN
		THIS^.addNewDispatcher(currentType);
		myCandyType := myCandyType XOR currentType;
		RETURN(myCandyType = 0);
	END_IF
END_FOR
END_METHOD

(*

short summary
=============
This message writes a ads log message if a consumer
was eating a concrete candy instance. The message
contains the consumer name, the amount, and the satisfaction
level of the consumer after the consume.

legal notes
===========
SPDX-FileCopyrightText: © 2024 ekvip automation GmbH <info@ekvip.de>
SPDX-License-Identifier: Apache-2.0
For details check: Apache-2.0_

.. _Apache-2.0: https://www.apache.org/licenses/LICENSE-2.0

*)
METHOD PROTECTED logCandyConsume
VAR_INPUT
	(* consumer who ate the candy *)
	consumer :REFERENCE TO AbstractCandyConsumer;
END_VAR
VAR
	(* format string because it's easier as the concatenation hell *)
	stringFromatter	:Tc2_Utilities.FB_FormatString;
	(* consumer name because we need a variable and not a property for the format string *)
	consumerName	:ConsumerName;
	(*
	satisfaction level of the consumer
	because we need a variable and not a property for the format string 
	*)
	statisfaction	:SatisfactionLevelInPercent;
END_VAR
VAR
	(* just a provider for a logger *)
	loggingProvider :LoggerProvider(0);
END_VAR
statisfaction := consumer.levelOfSatisfaction;
consumerName := consumer.name;
stringFromatter(
	sFormat := '%s was eating %d grams %s the satisfaction level of %s is now %d %%',
	arg1 := THIS^.anyToArg(consumerName),
	arg2 := THIS^.anyToArg(THIS^.amount),
	arg3 := THIS^.anyToArg(THIS^.name),
	arg4 := THIS^.anyToArg(consumerName),
	arg5 := THIS^.anyToArg(statisfaction),
);

loggingProvider.logger.info(stringFromatter.sOut);
END_METHOD

(*

short summary
=============
This property has just a getter, and it returns the
the name of the concrete candy like Snickers or Alpenliebe.

legal notes
===========
SPDX-FileCopyrightText: © 2024 ekvip automation GmbH <info@ekvip.de>
SPDX-License-Identifier: Apache-2.0
For details check: Apache-2.0_

.. _Apache-2.0: https://www.apache.org/licenses/LICENSE-2.0

*)
PROPERTY nameOfCandy : CandyName
GET
(*

short summary
=============
Just the getter for the name of the candy.

legal notes
===========
SPDX-FileCopyrightText: © 2024 ekvip automation GmbH <info@ekvip.de>
SPDX-License-Identifier: Apache-2.0
For details check: Apache-2.0_

.. _Apache-2.0: https://www.apache.org/licenses/LICENSE-2.0

*)
VAR
END_VAR
nameOfCandy := THIS^.name;
END_GET
END_PROPERTY

(*

short summary
=============
This property has just a getter, and it returns the
type of the candy. The type of the candy is a non-strict
enumeration because every candy type is represented by one
bit. For example a snickers is a candy bar, a caramel candy
and chocolate candy.

legal notes
===========
SPDX-FileCopyrightText: © 2024 ekvip automation GmbH <info@ekvip.de>
SPDX-License-Identifier: Apache-2.0
For details check: Apache-2.0_

.. _Apache-2.0: https://www.apache.org/licenses/LICENSE-2.0

*)
PROPERTY typeOfCandy :CandyTypes
GET
(*

short summary
=============
Just the getter for the type of candy.

legal notes
===========
SPDX-FileCopyrightText: © 2024 ekvip automation GmbH <info@ekvip.de>
SPDX-License-Identifier: Apache-2.0
For details check: Apache-2.0_

.. _Apache-2.0: https://www.apache.org/licenses/LICENSE-2.0

*)
VAR
END_VAR
typeOfCandy := THIS^.candyType;
END_GET
END_PROPERTY

END_FUNCTION_BLOCK

// ---- AnyToArg/Classes/AnyToTArgConverter.TcPOU
(*

short summary
=============
This abstract class provides a converter
form ANY type to the type Tc2_Utilities.T_Arg
Simply inherit from the class, then you can use the AnyToArg method.
This is much more convenient than the Tc2_Utilities.F_BYTE,
Tc2_Utilities.F_WORD etc. functions provided by Beckhoff.
The AnyToArg method is protected so it will not mess up your function block interface. 

legal notes
===========
SPDX-FileCopyrightText: © 2024 ekvip automation GmbH <info@ekvip.de>
SPDX-License-Identifier: Apache-2.0
For details check: Apache-2.0_

.. _Apache-2.0: https://www.apache.org/licenses/LICENSE-2.0

*)
FUNCTION_BLOCK ABSTRACT AnyToTArgConverter
VAR
END_VAR

(*

short summary
=============
This method takes an ANY type as input
parameter and returns a Tc2_Utilities.T_Arg of it.

legal notes
===========
SPDX-FileCopyrightText: © 2024 ekvip automation GmbH <info@ekvip.de>
SPDX-License-Identifier: Apache-2.0
For details check: Apache-2.0_

.. _Apache-2.0: https://www.apache.org/licenses/LICENSE-2.0

*)
METHOD PROTECTED FINAL anyToArg :Tc2_Utilities.T_Arg
VAR_INPUT
	(* just the data which shoud be casted to ``Tc2_Utilities.T_Arg`` *)
	in	:ANY;
END_VAR
VAR
	(* just to store the ``ANY`` without changes *)
	data	:__SYSTEM.AnyType;	
END_VAR
data.diSize := in.diSize;
data.pValue := in.pValue;
data.TypeClass := in.TypeClass;
THIS^.dereferenceAnys(in := data, out => data);
anyToArg := THIS^.anyTypeToArg(data);
END_METHOD

(*

short summary
=============
This method takes a __SYSTEM.AnyType type and returns a Tc2_Utilities.T_Arg of it.

legal notes
===========
SPDX-FileCopyrightText: © 2024 ekvip automation GmbH <info@ekvip.de>
SPDX-License-Identifier: Apache-2.0
For details check: Apache-2.0_

.. _Apache-2.0: https://www.apache.org/licenses/LICENSE-2.0

*)
METHOD PRIVATE anyTypeToArg :Tc2_Utilities.T_Arg
VAR_INPUT
	(* __SYSTEM.AnyType which should be converted to Tc2_Utilities.T_Arg *)
	in :__SYSTEM.AnyType;
END_VAR
anyTypeToArg.cbLen := TO_UDINT(in.diSize);
anyTypeToArg.pData := in.pValue;
anyTypeToArg.eType := THIS^.typeClassToArgType(in.TypeClass, anyTypeToArg.cbLen);
END_METHOD

(*

short summary
=============
This method is used to derference ANY types
until it find a non ANY type. The method is recursive.  

legal notes
===========
SPDX-FileCopyrightText: © 2024 ekvip automation GmbH <info@ekvip.de>
SPDX-License-Identifier: Apache-2.0
For details check: Apache-2.0_

.. _Apache-2.0: https://www.apache.org/licenses/LICENSE-2.0

*)
{attribute 'estimated-stack-usage' := '280'}
METHOD PRIVATE dereferenceAnys
VAR_INPUT
	(* __SYSTEM.AnyType to dereference *)
	in :__SYSTEM.AnyType;
END_VAR
VAR_OUTPUT
	(* dereferenced __SYSTEM.AnyType *)
	out :__SYSTEM.AnyType;	
END_VAR
VAR
	(* pointer to get the next address *)
	p :POINTER TO __SYSTEM.AnyType;
END_VAR
CASE in.TypeClass OF
__SYSTEM.TYPE_CLASS.TYPE_ANY,  
__SYSTEM.TYPE_CLASS.TYPE_ANYBIT, 
__SYSTEM.TYPE_CLASS.TYPE_ANYDATE,
__SYSTEM.TYPE_CLASS.TYPE_ANYINT,
__SYSTEM.TYPE_CLASS.TYPE_ANYNUM,
__SYSTEM.TYPE_CLASS.TYPE_ANYREAL:
	p := in.pValue;
	p := p^.pValue;
	THIS^.dereferenceAnys(p^, out => out);
ELSE
	out := in;
END_CASE
END_METHOD

(*

short summary
=============
This method translates the __SYSTEM.TYPE_CLASS form __SYSTEM.AnyType 
to Tc2_Utilities.E_ArgType from Tc2_Utilities.T_Arg

legal notes
===========
SPDX-FileCopyrightText: © 2024 ekvip automation GmbH <info@ekvip.de>
SPDX-License-Identifier: Apache-2.0
For details check: Apache-2.0_

.. _Apache-2.0: https://www.apache.org/licenses/LICENSE-2.0

*)
METHOD PRIVATE typeClassToArgType :Tc2_Utilities.E_ArgType
VAR_INPUT
	(* type class to translate *)
	typeClass :__SYSTEM.TYPE_CLASS;
	(* size to determine the base type *)
	size :UDINT;
END_VAR
CASE typeClass OF
__SYSTEM.TYPE_CLASS.TYPE_BOOL,
__SYSTEM.TYPE_CLASS.TYPE_BYTE,
__SYSTEM.TYPE_CLASS.TYPE_BIT,
__SYSTEM.TYPE_CLASS.TYPE_BITCONST:
	typeClassToArgType := Tc2_Utilities.E_ArgType.ARGTYPE_BYTE;
__SYSTEM.TYPE_CLASS.TYPE_WORD:
	typeClassToArgType := Tc2_Utilities.E_ArgType.ARGTYPE_WORD;
__SYSTEM.TYPE_CLASS.TYPE_DWORD:
	typeClassToArgType := Tc2_Utilities.E_ArgType.ARGTYPE_DWORD;
__SYSTEM.TYPE_CLASS.TYPE_LWORD:
	typeClassToArgType := Tc2_Utilities.E_ArgType.ARGTYPE_LWORD;
__SYSTEM.TYPE_CLASS.TYPE_USINT:
	typeClassToArgType := Tc2_Utilities.E_ArgType.ARGTYPE_USINT;
__SYSTEM.TYPE_CLASS.TYPE_SINT:
	typeClassToArgType := Tc2_Utilities.E_ArgType.ARGTYPE_SINT;
__SYSTEM.TYPE_CLASS.TYPE_UINT:
	typeClassToArgType := Tc2_Utilities.E_ArgType.ARGTYPE_UINT;
__SYSTEM.TYPE_CLASS.TYPE_INT:
	typeClassToArgType := Tc2_Utilities.E_ArgType.ARGTYPE_INT;
__SYSTEM.TYPE_CLASS.TYPE_UDINT, __SYSTEM.TYPE_CLASS.TYPE_TIME,
__SYSTEM.TYPE_CLASS.TYPE_DATE, __SYSTEM.TYPE_CLASS.TYPE_DATEANDTIME,
__SYSTEM.TYPE_CLASS.TYPE_TIMEOFDAY:
	typeClassToArgType := Tc2_Utilities.E_ArgType.ARGTYPE_UDINT;
__SYSTEM.TYPE_CLASS.TYPE_DINT:
	typeClassToArgType := Tc2_Utilities.E_ArgType.ARGTYPE_DINT;
__SYSTEM.TYPE_CLASS.TYPE_ULINT, __SYSTEM.TYPE_CLASS.TYPE_LTIME,
__SYSTEM.TYPE_CLASS.TYPE_LDATE, __SYSTEM.TYPE_CLASS.TYPE_LDATEANDTIME,
__SYSTEM.TYPE_CLASS.TYPE_LTIMEOFDAY:
		typeClassToArgType := Tc2_Utilities.E_ArgType.ARGTYPE_ULARGE;
__SYSTEM.TYPE_CLASS.TYPE_LINT:
	typeClassToArgType := Tc2_Utilities.E_ArgType.ARGTYPE_LARGE;
__SYSTEM.TYPE_CLASS.TYPE_XINT:
	typeClassToArgType := SEL(
		(SIZEOF(__XINT) = SIZEOF(LINT)),
		Tc2_Utilities.E_ArgType.ARGTYPE_DWORD,
		Tc2_Utilities.E_ArgType.ARGTYPE_LWORD
	);
__SYSTEM.TYPE_CLASS.TYPE_UXINT, __SYSTEM.TYPE_CLASS.TYPE_XWORD,
__SYSTEM.TYPE_CLASS.TYPE_POINTER, __SYSTEM.TYPE_CLASS.TYPE_REFERENCE:
	typeClassToArgType := SEL(
		(SIZEOF(__XWORD) = SIZEOF(LWORD)),
		Tc2_Utilities.E_ArgType.ARGTYPE_DWORD,
		Tc2_Utilities.E_ArgType.ARGTYPE_LWORD
	);	
__SYSTEM.TYPE_CLASS.TYPE_REAL:
	typeClassToArgType := Tc2_Utilities.E_ArgType.ARGTYPE_REAL;
__SYSTEM.TYPE_CLASS.TYPE_LREAL:
	typeClassToArgType := Tc2_Utilities.E_ArgType.ARGTYPE_LREAL;
__SYSTEM.TYPE_CLASS.TYPE_STRING:
	typeClassToArgType := SEL(
		(size <= SIZEOF(T_MaxString)),
		Tc2_Utilities.E_ArgType.ARGTYPE_BIGTYPE,
		Tc2_Utilities.E_ArgType.ARGTYPE_STRING
	);
__SYSTEM.TYPE_CLASS.TYPE_XSTRING:
{IF defined (NO_UNICODE_SUPPORT)}
	typeClassToArgType := SEL(
		(size <= SIZEOF(T_MaxString)),
		Tc2_Utilities.E_ArgType.ARGTYPE_BIGTYPE,
		Tc2_Utilities.E_ArgType.ARGTYPE_STRING
	);
{ELSE}
	typeClassToArgType := ARGTYPE_BIGTYPE;
{END_IF}
__SYSTEM.TYPE_CLASS.TYPE_WSTRING, __SYSTEM.TYPE_CLASS.TYPE_VARLENARRAY,
__SYSTEM.TYPE_CLASS.TYPE_USERDEF, __SYSTEM.TYPE_CLASS.TYPE_ARRAY,
__SYSTEM.TYPE_CLASS.TYPE_VECTOR:
	typeClassToArgType := ARGTYPE_BIGTYPE;	
__SYSTEM.TYPE_CLASS.TYPE_SUBRANGE, __SYSTEM.TYPE_CLASS.TYPE_ENUM:
	typeClassToArgType := MUX(
		size,
		(* size is 0 bytes *)
		Tc2_Utilities.E_ArgType.ARGTYPE_UNKNOWN,
		(* size is 1 bytes *)
		Tc2_Utilities.E_ArgType.ARGTYPE_SINT,
		(* size is 2 bytes *)
		Tc2_Utilities.E_ArgType.ARGTYPE_INT,
		(* size is 3 bytes *)
		Tc2_Utilities.E_ArgType.ARGTYPE_UNKNOWN,
		(* size is 4 bytes *)
		Tc2_Utilities.E_ArgType.ARGTYPE_DINT,
		(* size is 5 bytes *)
		Tc2_Utilities.E_ArgType.ARGTYPE_UNKNOWN,
		(* size is 6 bytes *)
		Tc2_Utilities.E_ArgType.ARGTYPE_UNKNOWN,
		(* size is 7 bytes *)
		Tc2_Utilities.E_ArgType.ARGTYPE_UNKNOWN,
		(* size is 8 bytes *)
		Tc2_Utilities.E_ArgType.ARGTYPE_ULARGE,
		(* size is more than 8 bytes *)
		Tc2_Utilities.E_ArgType.ARGTYPE_BIGTYPE
	);
__SYSTEM.TYPE_CLASS.TYPE_LAZY,
__SYSTEM.TYPE_CLASS.TYPE_NONE,
__SYSTEM.TYPE_CLASS.TYPE_PARAMS:
	typeClassToArgType := Tc2_Utilities.E_ArgType.ARGTYPE_UNKNOWN;
ELSE
	typeClassToArgType := Tc2_Utilities.E_ArgType.ARGTYPE_UNKNOWN;
END_CASE
END_METHOD

END_FUNCTION_BLOCK

// ---- CandyDispatchers/Classes/AbstractCandyDispatcher.TcPOU
(*

short summary
=============
dispatcher to unify the eat<CandyType> method call of the candy consumer.
It's just annoying to call for every candy types differnt methods.
It is possible to use the same code to dispatch the candy to the
consumer. We just delegate it to the right dispatcher.
Every candy will creacte the required dispatcher dynamicly in the
class AbstactCandy in the method initializeDispatchers.

legal notes
===========
SPDX-FileCopyrightText: © 2024 ekvip automation GmbH <info@ekvip.de>
SPDX-License-Identifier: Apache-2.0
For details check: Apache-2.0_

.. _Apache-2.0: https://www.apache.org/licenses/LICENSE-2.0

*)

FUNCTION_BLOCK ABSTRACT AbstractCandyDispatcher

(*

short summary
=============
This method is to free the memory again 
if the dispatcher was created dynamicly.
It's easier to provide this method than
to __querypointer until it matches.

legal notes
===========
SPDX-FileCopyrightText: © 2024 ekvip automation GmbH <info@ekvip.de>
SPDX-License-Identifier: Apache-2.0
For details check: Apache-2.0_

.. _Apache-2.0: https://www.apache.org/licenses/LICENSE-2.0

*)

METHOD destruct :POINTER TO AbstractCandyDispatcher
VAR_INPUT
END_VAR
VAR CONSTANT
	(* just null pointer as return value *)
	NULL :__XWORD := 0;
END_VAR
destruct := THIS;
IF (
	Tc2_System.F_CheckMemoryArea(pData := THIS, nSize := SIZEOF(THIS^))
	= Tc2_System.E_TcMemoryArea.Dynamic
) THEN
	__DELETE(destruct);
	destruct := NULL;
END_IF
END_METHOD

(*

short summary
=============
this is the method to unify the
counsumers eat what erver calls 

legal notes
===========
SPDX-FileCopyrightText: © 2024 ekvip automation GmbH <info@ekvip.de>
SPDX-License-Identifier: Apache-2.0
For details check: Apache-2.0_

.. _Apache-2.0: https://www.apache.org/licenses/LICENSE-2.0

*)

METHOD ABSTRACT eat
VAR_INPUT
	(* consumer who eats the candy *)
	consumer	:REFERENCE TO AbstractCandyConsumer;
	(* candy amount in gram *)
	amount		:CandyAmountInGram;
END_VAR
END_METHOD

(*

short summary
=============
just a helper to test the parameters
- it returns true if minimum one of the parameters is invalid
- it retruns false if all parameters are valid

legal notes
===========
SPDX-FileCopyrightText: © 2024 ekvip automation GmbH <info@ekvip.de>
SPDX-License-Identifier: Apache-2.0
For details check: Apache-2.0_

.. _Apache-2.0: https://www.apache.org/licenses/LICENSE-2.0

*)

METHOD PROTECTED eatCandiesIsImpossible :BOOL
VAR_INPUT
	(* consumer who eats the candy *)
	consumer	:REFERENCE TO AbstractCandyConsumer;
	(* candy amount in gram *)
	amount		:CandyAmountInGram;
END_VAR
eatCandiesIsImpossible := TRUE;
RETURN(NOT __ISVALIDREF(consumer));
RETURN(amount <= 0);
eatCandiesIsImpossible := FALSE;
END_METHOD

END_FUNCTION_BLOCK

// ---- CandyConsumer/Classes/AbstractCandyConsumer.TcPOU
(*

short summary
=============
A candy consumer. It can eat candies and the
candies will effect the satisfaction of the consumer.  

legal notes
===========
SPDX-FileCopyrightText: © 2024 ekvip automation GmbH <info@ekvip.de>
SPDX-License-Identifier: Apache-2.0
For details check: Apache-2.0_

.. _Apache-2.0: https://www.apache.org/licenses/LICENSE-2.0

*)

FUNCTION_BLOCK ABSTRACT AbstractCandyConsumer
VAR
	(* the satisfaction level of the consumer in % *)
	satisfaction :SatisfactionLevelInPercent;
END_VAR

(*

short summary
=============
method to eat candy bars

legal notes
===========
SPDX-FileCopyrightText: © 2024 ekvip automation GmbH <info@ekvip.de>
SPDX-License-Identifier: Apache-2.0
For details check: Apache-2.0_

.. _Apache-2.0: https://www.apache.org/licenses/LICENSE-2.0

*)

METHOD ABSTRACT eatCandyBars
VAR_INPUT
	(* amount of candy that the consumer eats in gram *)
	amount	:CandyAmountInGram;
END_VAR
END_METHOD

(*

short summary
=============
method to eat candy corn

legal notes
===========
SPDX-FileCopyrightText: © 2024 ekvip automation GmbH <info@ekvip.de>
SPDX-License-Identifier: Apache-2.0
For details check: Apache-2.0_

.. _Apache-2.0: https://www.apache.org/licenses/LICENSE-2.0

*)

METHOD ABSTRACT eatCandyCorn
VAR_INPUT
	(* amount of candy that the consumer eats in gram *)
	amount	:CandyAmountInGram;
END_VAR
END_METHOD

(*

short summary
=============
method to eat candy sticks

legal notes
===========
SPDX-FileCopyrightText: © 2024 ekvip automation GmbH <info@ekvip.de>
SPDX-License-Identifier: Apache-2.0
For details check: Apache-2.0_

.. _Apache-2.0: https://www.apache.org/licenses/LICENSE-2.0

*)

METHOD ABSTRACT eatCandySticks
VAR_INPUT
	(* amount of candy that the consumer eats in gram *)
	amount	:CandyAmountInGram;
END_VAR
END_METHOD

(*

short summary
=============
method to eat caramel candy

legal notes
===========
SPDX-FileCopyrightText: © 2024 ekvip automation GmbH <info@ekvip.de>
SPDX-License-Identifier: Apache-2.0
For details check: Apache-2.0_

.. _Apache-2.0: https://www.apache.org/licenses/LICENSE-2.0

*)

METHOD ABSTRACT eatCaramelCandy
VAR_INPUT
	(* amount of candy that the consumer eats in gram *)
	amount	:CandyAmountInGram;
END_VAR
END_METHOD

(*

short summary
=============
method to eat choclate candy

legal notes
===========
SPDX-FileCopyrightText: © 2024 ekvip automation GmbH <info@ekvip.de>
SPDX-License-Identifier: Apache-2.0
For details check: Apache-2.0_

.. _Apache-2.0: https://www.apache.org/licenses/LICENSE-2.0

*)

METHOD ABSTRACT eatChoclateCandy
VAR_INPUT
	(* amount of candy that the consumer eats in gram *)
	amount	:CandyAmountInGram;
END_VAR
END_METHOD

(*

short summary
=============
method to eat gummy candy

legal notes
===========
SPDX-FileCopyrightText: © 2024 ekvip automation GmbH <info@ekvip.de>
SPDX-License-Identifier: Apache-2.0
For details check: Apache-2.0_

.. _Apache-2.0: https://www.apache.org/licenses/LICENSE-2.0

*)

METHOD ABSTRACT eatGummyCandy
VAR_INPUT
	(* amount of candy that the consumer eats in gram *)
	amount	:CandyAmountInGram;
END_VAR
END_METHOD

(*

short summary
=============
method to eat hard candy

legal notes
===========
SPDX-FileCopyrightText: © 2024 ekvip automation GmbH <info@ekvip.de>
SPDX-License-Identifier: Apache-2.0
For details check: Apache-2.0_

.. _Apache-2.0: https://www.apache.org/licenses/LICENSE-2.0

*)

METHOD ABSTRACT eatHardCandy
VAR_INPUT
	(* amount of candy that the consumer eats in gram *)
	amount	:CandyAmountInGram;
END_VAR
END_METHOD

(*

short summary
=============
method to eat jawbreakers

legal notes
===========
SPDX-FileCopyrightText: © 2024 ekvip automation GmbH <info@ekvip.de>
SPDX-License-Identifier: Apache-2.0
For details check: Apache-2.0_

.. _Apache-2.0: https://www.apache.org/licenses/LICENSE-2.0

*)

METHOD ABSTRACT eatJawbreakers
VAR_INPUT
	(* amount of candy that the consumer eats in gram *)
	amount	:CandyAmountInGram;
END_VAR
END_METHOD

(*

short summary
=============
method to eat licorice candy

legal notes
===========
SPDX-FileCopyrightText: © 2024 ekvip automation GmbH <info@ekvip.de>
SPDX-License-Identifier: Apache-2.0
For details check: Apache-2.0_

.. _Apache-2.0: https://www.apache.org/licenses/LICENSE-2.0

*)

METHOD ABSTRACT eatLicoriceCandy
VAR_INPUT
	(* amount of candy that the consumer eats in gram *)
	amount	:CandyAmountInGram;
END_VAR
END_METHOD

(*

short summary
=============
method to eat lollipops

legal notes
===========
SPDX-FileCopyrightText: © 2024 ekvip automation GmbH <info@ekvip.de>
SPDX-License-Identifier: Apache-2.0
For details check: Apache-2.0_

.. _Apache-2.0: https://www.apache.org/licenses/LICENSE-2.0

*)

METHOD ABSTRACT eatLollipops
VAR_INPUT
	(* amount of candy that the consumer eats in gram *)
	amount	:CandyAmountInGram;
END_VAR
END_METHOD

(*

short summary
=============
method to eat mints

legal notes
===========
SPDX-FileCopyrightText: © 2024 ekvip automation GmbH <info@ekvip.de>
SPDX-License-Identifier: Apache-2.0
For details check: Apache-2.0_

.. _Apache-2.0: https://www.apache.org/licenses/LICENSE-2.0

*)

METHOD ABSTRACT eatMints
VAR_INPUT
	(* amount of candy that the consumer eats in gram *)
	amount	:CandyAmountInGram;
END_VAR
END_METHOD

(*

short summary
=============
method to eat sour candy

legal notes
===========
SPDX-FileCopyrightText: © 2024 ekvip automation GmbH <info@ekvip.de>
SPDX-License-Identifier: Apache-2.0
For details check: Apache-2.0_

.. _Apache-2.0: https://www.apache.org/licenses/LICENSE-2.0

*)

METHOD ABSTRACT eatSourCandy
VAR_INPUT
	(* amount of candy that the consumer eats in gram *)
	amount	:CandyAmountInGram;
END_VAR
END_METHOD

(*

short summary
=============
The actual satisfaction level of the consumer
in percent 0% means depression 100% means euphoria
The consumer has just a getter for the satisfaction level

legal notes
===========
SPDX-FileCopyrightText: © 2024 ekvip automation GmbH <info@ekvip.de>
SPDX-License-Identifier: Apache-2.0
For details check: Apache-2.0_

.. _Apache-2.0: https://www.apache.org/licenses/LICENSE-2.0

*)

PROPERTY levelOfSatisfaction :SatisfactionLevelInPercent
GET
(*

short summary
=============
Getter for the actual satisfaction level of the consumer
in percent 0% means depression 100% means euphoria.

legal notes
===========
SPDX-FileCopyrightText: © 2024 ekvip automation GmbH <info@ekvip.de>
SPDX-License-Identifier: Apache-2.0
For details check: Apache-2.0_

.. _Apache-2.0: https://www.apache.org/licenses/LICENSE-2.0

*)

VAR
END_VAR
levelOfSatisfaction := THIS^.satisfaction;
END_GET
END_PROPERTY

(*

short summary
=============
name of the consumer

legal notes
===========
SPDX-FileCopyrightText: © 2024 ekvip automation GmbH <info@ekvip.de>
SPDX-License-Identifier: Apache-2.0
For details check: Apache-2.0_

.. _Apache-2.0: https://www.apache.org/licenses/LICENSE-2.0

*)

PROPERTY ABSTRACT name :ConsumerName
GET
(*

short summary
=============
getter for the name of the consumer
for logging purpose

legal notes
===========
SPDX-FileCopyrightText: © 2024 ekvip automation GmbH <info@ekvip.de>
SPDX-License-Identifier: Apache-2.0
For details check: Apache-2.0_

.. _Apache-2.0: https://www.apache.org/licenses/LICENSE-2.0

*)

VAR
END_VAR
END_GET
END_PROPERTY

END_FUNCTION_BLOCK

// ---- CandyDispatchers/Classes/CandyDispatcherFactory.TcPOU
(*

short summary
=============
factory class to create new 
dispatcher according to the candy type

legal notes
===========
SPDX-FileCopyrightText: © 2024 ekvip automation GmbH <info@ekvip.de>
SPDX-License-Identifier: Apache-2.0
For details check: Apache-2.0_

.. _Apache-2.0: https://www.apache.org/licenses/LICENSE-2.0

*)

FUNCTION_BLOCK FINAL CandyDispatcherFactory

(*

short summary
=============
method creates a new dispatcher instance
for a given candy type, but it must be a 
pure candy type. To free the memory again
use the destruct method of the dispatcher.

legal notes
===========
SPDX-FileCopyrightText: © 2024 ekvip automation GmbH <info@ekvip.de>
SPDX-License-Identifier: Apache-2.0
For details check: Apache-2.0_

.. _Apache-2.0: https://www.apache.org/licenses/LICENSE-2.0

*)

METHOD getNewCandyDispatcherFor :POINTER TO AbstractCandyDispatcher
VAR_INPUT
	(* candy type to create the right dispatcher, it must be a pure candy type *) 
	candyType	:CandyTypes;
END_VAR
VAR
	(* the __NEW operator requires a stricktly typed pointer *)
	candyBarDelegator		:POINTER TO CandyBarDispatcher;
	(* the __NEW operator requires a stricktly typed pointer *)
	candyCornDelegator		:POINTER TO CandyCornDispatcher;
	(* the __NEW operator requires a stricktly typed pointer *)
	candySticksDelegator	:POINTER TO CandySticksDispatcher; 
	(* the __NEW operator requires a stricktly typed pointer *)
	caramelCandyDelegator	:POINTER TO CaramelCandyDispatcher;
	(* the __NEW operator requires a stricktly typed pointer *)
	chocolateCandyDelegator	:POINTER TO ChoclateCandyDispatcher;
	(* the __NEW operator requires a stricktly typed pointer *)
	gummyCandyDelegator		:POINTER TO GummyCandyDispatcher;
	(* the __NEW operator requires a stricktly typed pointer *)
	mintsDelegator			:POINTER TO MintsDispatcher;
	(* the __NEW operator requires a stricktly typed pointer *)
	lolliposDelegator		:POINTER TO LollipopsDispatcher;
	(* the __NEW operator requires a stricktly typed pointer *)
	jawbreakersDelegator	:POINTER TO JawbreakersDispatcher; 
	(* the __NEW operator requires a stricktly typed pointer *)
	hardCandyDelegator		:POINTER TO HardCandyDispatcher;
	(* the __NEW operator requires a stricktly typed pointer *)
	licoriceDelegator		:POINTER TO LicoriceCandyDispatcher;
	(* the __NEW operator requires a stricktly typed pointer *)
	sourCandyDelegator		:POINTER TO SourCandyDispatcher;
END_VAR
getNewCandyDispatcherFor := 0;
CASE candyType OF
CandyTypes.CANDY_BARS:
	candyBarDelegator := __NEW(CandyBarDispatcher());
	getNewCandyDispatcherFor := candyBarDelegator;
CandyTypes.CANDY_CORN:
	candyCornDelegator := __NEW(CandyCornDispatcher());
	getNewCandyDispatcherFor := candyCornDelegator;
CandyTypes.CANDY_STICKS:
	candySticksDelegator := __NEW(CandySticksDispatcher());
	getNewCandyDispatcherFor := candySticksDelegator;	
CandyTypes.CARAMEL_CANDY:
	caramelCandyDelegator := __NEW(CaramelCandyDispatcher());
	getNewCandyDispatcherFor := caramelCandyDelegator;	
CandyTypes.CHOCOLATE_CANDY:
	chocolateCandyDelegator := __NEW(ChoclateCandyDispatcher());
	getNewCandyDispatcherFor := chocolateCandyDelegator;	
CandyTypes.GUMMY_CANDY:
	gummyCandyDelegator := __NEW(GummyCandyDispatcher());
	getNewCandyDispatcherFor := gummyCandyDelegator;	
CandyTypes.HARD_CANDY:
	hardCandyDelegator := __NEW(HardCandyDispatcher());
	getNewCandyDispatcherFor := hardCandyDelegator;	
CandyTypes.JAWBREAKERS:
	jawbreakersDelegator := __NEW(JawbreakersDispatcher());
	getNewCandyDispatcherFor := jawbreakersDelegator;	
CandyTypes.LICORICE_CANDY:
	licoriceDelegator := __NEW(LicoriceCandyDispatcher());
	getNewCandyDispatcherFor := licoriceDelegator;	
CandyTypes.LOLLIPOPS:
	lolliposDelegator := __NEW(LollipopsDispatcher());
	getNewCandyDispatcherFor := lolliposDelegator;	
CandyTypes.MINTS:
	mintsDelegator := __NEW(MintsDispatcher());
	getNewCandyDispatcherFor := mintsDelegator;
CandyTypes.SOUR_CANDY:
	sourCandyDelegator := __NEW(SourCandyDispatcher());
	getNewCandyDispatcherFor := sourCandyDelegator;
ELSE
	RETURN;
END_CASE
END_METHOD

END_FUNCTION_BLOCK

// ---- CandyDispatchers/Classes/CandyBarDispatcher.TcPOU
(*

short summary
=============
dispather for candy bars

legal notes
===========
SPDX-FileCopyrightText: © 2024 ekvip automation GmbH <info@ekvip.de>
SPDX-License-Identifier: Apache-2.0
For details check: Apache-2.0_

.. _Apache-2.0: https://www.apache.org/licenses/LICENSE-2.0

*)

{attribute 'enable_dynamic_creation'}
FUNCTION_BLOCK FINAL CandyBarDispatcher EXTENDS AbstractCandyDispatcher

(*

short summary
=============
this method dispatches candy bars
to a candy consumer 

legal notes
===========
SPDX-FileCopyrightText: © 2024 ekvip automation GmbH <info@ekvip.de>
SPDX-License-Identifier: Apache-2.0
For details check: Apache-2.0_

.. _Apache-2.0: https://www.apache.org/licenses/LICENSE-2.0

*)

METHOD eat
VAR_INPUT
	(* consumer who eats the candy *)
	consumer	:REFERENCE TO AbstractCandyConsumer;
	(* candy amount in gram *)
	amount		:CandyAmountInGram;
END_VAR
RETURN(THIS^.eatCandiesIsImpossible(consumer, amount));
consumer.eatCandyBars(amount);
END_METHOD

END_FUNCTION_BLOCK

// ---- CandyDispatchers/Classes/CandyCornDispatcher.TcPOU
(*

short summary
=============
dispather for candy corn

legal notes
===========
SPDX-FileCopyrightText: © 2024 ekvip automation GmbH <info@ekvip.de>
SPDX-License-Identifier: Apache-2.0
For details check: Apache-2.0_

.. _Apache-2.0: https://www.apache.org/licenses/LICENSE-2.0

*)

{attribute 'enable_dynamic_creation'}
FUNCTION_BLOCK FINAL CandyCornDispatcher EXTENDS AbstractCandyDispatcher

(*

short summary
=============
this method dispatches candy corn
to a candy consumer 

legal notes
===========
SPDX-FileCopyrightText: © 2024 ekvip automation GmbH <info@ekvip.de>
SPDX-License-Identifier: Apache-2.0
For details check: Apache-2.0_

.. _Apache-2.0: https://www.apache.org/licenses/LICENSE-2.0

*)

METHOD eat
VAR_INPUT
	(* consumer who eats the candy *)
	consumer	:REFERENCE TO AbstractCandyConsumer;
	(* candy amount in gram *)
	amount		:CandyAmountInGram;
END_VAR
RETURN(THIS^.eatCandiesIsImpossible(consumer, amount));
consumer.eatCandyCorn(amount);
END_METHOD

END_FUNCTION_BLOCK

// ---- CandyDispatchers/Classes/CandySticksDispatcher.TcPOU
(*

short summary
=============
dispather for candy sticks

legal notes
===========
SPDX-FileCopyrightText: © 2024 ekvip automation GmbH <info@ekvip.de>
SPDX-License-Identifier: Apache-2.0
For details check: Apache-2.0_

.. _Apache-2.0: https://www.apache.org/licenses/LICENSE-2.0

*)

{attribute 'enable_dynamic_creation'}
FUNCTION_BLOCK FINAL CandySticksDispatcher EXTENDS AbstractCandyDispatcher

(*

short summary
=============
this method dispatches candy sticks
to a candy consumer 

legal notes
===========
SPDX-FileCopyrightText: © 2024 ekvip automation GmbH <info@ekvip.de>
SPDX-License-Identifier: Apache-2.0
For details check: Apache-2.0_

.. _Apache-2.0: https://www.apache.org/licenses/LICENSE-2.0

*)

METHOD eat
VAR_INPUT
	(* consumer who eats the candy *)
	consumer	:REFERENCE TO AbstractCandyConsumer;
	(* candy amount in gram *)
	amount		:CandyAmountInGram;
END_VAR
RETURN(THIS^.eatCandiesIsImpossible(consumer, amount));
consumer.eatCandySticks(amount);
END_METHOD

END_FUNCTION_BLOCK

// ---- CandyDispatchers/Classes/CaramelCandyDispatcher.TcPOU
(*

short summary
=============
dispather for cramel candy

legal notes
===========
SPDX-FileCopyrightText: © 2024 ekvip automation GmbH <info@ekvip.de>
SPDX-License-Identifier: Apache-2.0
For details check: Apache-2.0_

.. _Apache-2.0: https://www.apache.org/licenses/LICENSE-2.0

*)

{attribute 'enable_dynamic_creation'}
FUNCTION_BLOCK FINAL CaramelCandyDispatcher EXTENDS AbstractCandyDispatcher

(*

short summary
=============
this method dispatches caramel candies
to a candy consumer 

legal notes
===========
SPDX-FileCopyrightText: © 2024 ekvip automation GmbH <info@ekvip.de>
SPDX-License-Identifier: Apache-2.0
For details check: Apache-2.0_

.. _Apache-2.0: https://www.apache.org/licenses/LICENSE-2.0

*)

METHOD eat
VAR_INPUT
	(* consumer who eats the candy *)
	consumer	:REFERENCE TO AbstractCandyConsumer;
	(* candy amount in gram *)
	amount		:CandyAmountInGram;
END_VAR
RETURN(THIS^.eatCandiesIsImpossible(consumer, amount));
consumer.eatCaramelCandy(amount);
END_METHOD

END_FUNCTION_BLOCK

// ---- CandyDispatchers/Classes/ChoclateCandyDispatcher.TcPOU
(*

short summary
=============
dispather for choclate candy

legal notes
===========
SPDX-FileCopyrightText: © 2024 ekvip automation GmbH <info@ekvip.de>
SPDX-License-Identifier: Apache-2.0
For details check: Apache-2.0_

.. _Apache-2.0: https://www.apache.org/licenses/LICENSE-2.0

*)

{attribute 'enable_dynamic_creation'}
FUNCTION_BLOCK FINAL ChoclateCandyDispatcher EXTENDS AbstractCandyDispatcher

(*

short summary
=============
this method dispatches choclate candies
to a candy consumer 

legal notes
===========
SPDX-FileCopyrightText: © 2024 ekvip automation GmbH <info@ekvip.de>
SPDX-License-Identifier: Apache-2.0
For details check: Apache-2.0_

.. _Apache-2.0: https://www.apache.org/licenses/LICENSE-2.0

*)

METHOD eat
VAR_INPUT
	(* consumer who eats the candy *)
	consumer	:REFERENCE TO AbstractCandyConsumer;
	(* candy amount in gram *)
	amount		:CandyAmountInGram;
END_VAR
RETURN(THIS^.eatCandiesIsImpossible(consumer, amount));
consumer.eatChoclateCandy(amount);
END_METHOD

END_FUNCTION_BLOCK

// ---- CandyDispatchers/Classes/GummyCandyDispatcher.TcPOU
(*

short summary
=============
dispather for gummy candy

legal notes
===========
SPDX-FileCopyrightText: © 2024 ekvip automation GmbH <info@ekvip.de>
SPDX-License-Identifier: Apache-2.0
For details check: Apache-2.0_

.. _Apache-2.0: https://www.apache.org/licenses/LICENSE-2.0

*)

{attribute 'enable_dynamic_creation'}
FUNCTION_BLOCK FINAL GummyCandyDispatcher EXTENDS AbstractCandyDispatcher

(*

short summary
=============
this method dispatches gummy candies
to a candy consumer 

legal notes
===========
SPDX-FileCopyrightText: © 2024 ekvip automation GmbH <info@ekvip.de>
SPDX-License-Identifier: Apache-2.0
For details check: Apache-2.0_

.. _Apache-2.0: https://www.apache.org/licenses/LICENSE-2.0

*)

METHOD eat
VAR_INPUT
	(* consumer who eats the candy *)
	consumer	:REFERENCE TO AbstractCandyConsumer;
	(* candy amount in gram *)
	amount		:CandyAmountInGram;
END_VAR
RETURN(THIS^.eatCandiesIsImpossible(consumer, amount));
consumer.eatGummyCandy(amount);
END_METHOD

END_FUNCTION_BLOCK

// ---- CandyDispatchers/Classes/MintsDispatcher.TcPOU
(*

short summary
=============
dispather for mints

legal notes
===========
SPDX-FileCopyrightText: © 2024 ekvip automation GmbH <info@ekvip.de>
SPDX-License-Identifier: Apache-2.0
For details check: Apache-2.0_

.. _Apache-2.0: https://www.apache.org/licenses/LICENSE-2.0

*)

{attribute 'enable_dynamic_creation'}
FUNCTION_BLOCK FINAL MintsDispatcher EXTENDS AbstractCandyDispatcher

(*

short summary
=============
this method dispatches mints
to a candy consumer 

legal notes
===========
SPDX-FileCopyrightText: © 2024 ekvip automation GmbH <info@ekvip.de>
SPDX-License-Identifier: Apache-2.0
For details check: Apache-2.0_

.. _Apache-2.0: https://www.apache.org/licenses/LICENSE-2.0

*)

METHOD eat
VAR_INPUT
	(* consumer who eats the candy *)
	consumer	:REFERENCE TO AbstractCandyConsumer;
	(* candy amount in gram *)
	amount		:CandyAmountInGram;
END_VAR
RETURN(THIS^.eatCandiesIsImpossible(consumer, amount));
consumer.eatMints(amount);
END_METHOD

END_FUNCTION_BLOCK

// ---- CandyDispatchers/Classes/LollipopsDispatcher.TcPOU
(*

short summary
=============
dispather for lollipops

legal notes
===========
SPDX-FileCopyrightText: © 2024 ekvip automation GmbH <info@ekvip.de>
SPDX-License-Identifier: Apache-2.0
For details check: Apache-2.0_

.. _Apache-2.0: https://www.apache.org/licenses/LICENSE-2.0

*)

{attribute 'enable_dynamic_creation'}
FUNCTION_BLOCK FINAL LollipopsDispatcher EXTENDS AbstractCandyDispatcher

(*

short summary
=============
this method dispatches lollipops
to a candy consumer 

legal notes
===========
SPDX-FileCopyrightText: © 2024 ekvip automation GmbH <info@ekvip.de>
SPDX-License-Identifier: Apache-2.0
For details check: Apache-2.0_

.. _Apache-2.0: https://www.apache.org/licenses/LICENSE-2.0

*)

METHOD eat
VAR_INPUT
	(* consumer who eats the candy *)
	consumer	:REFERENCE TO AbstractCandyConsumer;
	(* candy amount in gram *)
	amount		:CandyAmountInGram;
END_VAR
RETURN(THIS^.eatCandiesIsImpossible(consumer, amount));
consumer.eatLollipops(amount);
END_METHOD

END_FUNCTION_BLOCK

// ---- CandyDispatchers/Classes/JawbreakersDispatcher.TcPOU
(*

short summary
=============
dispather for jawbreakers

legal notes
===========
SPDX-FileCopyrightText: © 2024 ekvip automation GmbH <info@ekvip.de>
SPDX-License-Identifier: Apache-2.0
For details check: Apache-2.0_

.. _Apache-2.0: https://www.apache.org/licenses/LICENSE-2.0

*)

{attribute 'enable_dynamic_creation'}
FUNCTION_BLOCK FINAL JawbreakersDispatcher EXTENDS AbstractCandyDispatcher

(*

short summary
=============
this method dispatches jawbreakers
to a candy consumer 

legal notes
===========
SPDX-FileCopyrightText: © 2024 ekvip automation GmbH <info@ekvip.de>
SPDX-License-Identifier: Apache-2.0
For details check: Apache-2.0_

.. _Apache-2.0: https://www.apache.org/licenses/LICENSE-2.0

*)

METHOD  eat
VAR_INPUT
	(* consumer who eats the candy *)
	consumer	:REFERENCE TO AbstractCandyConsumer;
	(* candy amount in gram *)
	amount		:CandyAmountInGram;
END_VAR
RETURN(THIS^.eatCandiesIsImpossible(consumer, amount));
consumer.eatJawbreakers(amount);
END_METHOD

END_FUNCTION_BLOCK

// ---- CandyDispatchers/Classes/HardCandyDispatcher.TcPOU
(*

short summary
=============
dispather for hard candy

legal notes
===========
SPDX-FileCopyrightText: © 2024 ekvip automation GmbH <info@ekvip.de>
SPDX-License-Identifier: Apache-2.0
For details check: Apache-2.0_

.. _Apache-2.0: https://www.apache.org/licenses/LICENSE-2.0

*)

{attribute 'enable_dynamic_creation'}
FUNCTION_BLOCK FINAL HardCandyDispatcher EXTENDS AbstractCandyDispatcher

(*

short summary
=============
this method dispatches hard candies
to a candy consumer 

legal notes
===========
SPDX-FileCopyrightText: © 2024 ekvip automation GmbH <info@ekvip.de>
SPDX-License-Identifier: Apache-2.0
For details check: Apache-2.0_

.. _Apache-2.0: https://www.apache.org/licenses/LICENSE-2.0

*)

METHOD eat
VAR_INPUT
	(* consumer who eats the candy *)
	consumer	:REFERENCE TO AbstractCandyConsumer;
	(* candy amount in gram *)
	amount		:CandyAmountInGram;
END_VAR
RETURN(THIS^.eatCandiesIsImpossible(consumer, amount));
consumer.eatHardCandy(amount);
END_METHOD

END_FUNCTION_BLOCK

// ---- CandyDispatchers/Classes/LicoriceCandyDispatcher.TcPOU
(*

short summary
=============
dispather for licorice candy

legal notes
===========
SPDX-FileCopyrightText: © 2024 ekvip automation GmbH <info@ekvip.de>
SPDX-License-Identifier: Apache-2.0
For details check: Apache-2.0_

.. _Apache-2.0: https://www.apache.org/licenses/LICENSE-2.0

*)

{attribute 'enable_dynamic_creation'}
FUNCTION_BLOCK FINAL LicoriceCandyDispatcher EXTENDS AbstractCandyDispatcher

(*

short summary
=============
this method dispatches licorice candies
to a candy consumer 

legal notes
===========
SPDX-FileCopyrightText: © 2024 ekvip automation GmbH <info@ekvip.de>
SPDX-License-Identifier: Apache-2.0
For details check: Apache-2.0_

.. _Apache-2.0: https://www.apache.org/licenses/LICENSE-2.0

*)

METHOD eat
VAR_INPUT
	(* consumer who eats the candy *)
	consumer	:REFERENCE TO AbstractCandyConsumer;
	(* candy amount in gram *)
	amount		:CandyAmountInGram;
END_VAR
RETURN(THIS^.eatCandiesIsImpossible(consumer, amount));
consumer.eatLicoriceCandy(amount);
END_METHOD

END_FUNCTION_BLOCK

// ---- CandyDispatchers/Classes/SourCandyDispatcher.TcPOU
(*

short summary
=============
dispather for sour candy

legal notes
===========
SPDX-FileCopyrightText: © 2024 ekvip automation GmbH <info@ekvip.de>
SPDX-License-Identifier: Apache-2.0
For details check: Apache-2.0_

.. _Apache-2.0: https://www.apache.org/licenses/LICENSE-2.0

*)

{attribute 'enable_dynamic_creation'}
FUNCTION_BLOCK FINAL SourCandyDispatcher EXTENDS AbstractCandyDispatcher

(*

short summary
=============
this method dispatches sour candies
to a candy consumer 

legal notes
===========
SPDX-FileCopyrightText: © 2024 ekvip automation GmbH <info@ekvip.de>
SPDX-License-Identifier: Apache-2.0
For details check: Apache-2.0_

.. _Apache-2.0: https://www.apache.org/licenses/LICENSE-2.0

*)

METHOD eat
VAR_INPUT
	(* consumer who eats the candy *)
	consumer	:REFERENCE TO AbstractCandyConsumer;
	(* candy amount in gram *)
	amount		:CandyAmountInGram;
END_VAR
RETURN(THIS^.eatCandiesIsImpossible(consumer, amount));
consumer.eatSourCandy(amount);
END_METHOD

END_FUNCTION_BLOCK

// ---- CandyMachine/Classes/CommonCandyMachine.TcPOU
(*

short summary
=============
a candy vending machine for the usual eaters.

legal notes
===========
SPDX-FileCopyrightText: © 2024 ekvip automation GmbH <info@ekvip.de>
SPDX-License-Identifier: Apache-2.0
For details check: Apache-2.0_

.. _Apache-2.0: https://www.apache.org/licenses/LICENSE-2.0

*)

FUNCTION_BLOCK FINAL CommonCandyMachine EXTENDS AbstractCandyMachine

(*

short summary
=============
want some, get some
this method provides the candies

legal notes
===========
SPDX-FileCopyrightText: © 2024 ekvip automation GmbH <info@ekvip.de>
SPDX-License-Identifier: Apache-2.0
For details check: Apache-2.0_

.. _Apache-2.0: https://www.apache.org/licenses/LICENSE-2.0

*)

METHOD  getNewCandy :REFERENCE TO AbstractCandy
VAR_INPUT
	(*preferred candy type, it must be a pure candy type *)
	candyType	:CandyTypes;
END_VAR
VAR
	(* the __NEW operator requires a stricktly typed pointer *)
	altoids				:POINTER TO Altoids;
	(* the __NEW operator requires a stricktly typed pointer *)
	bobsStripes			:POINTER TO BobsSweetStripes;
	(* the __NEW operator requires a stricktly typed pointer *)
	candyCorn			:POINTER TO BrachsCandyCorn;
	(* the __NEW operator requires a stricktly typed pointer *)
	chupChups			:POINTER TO ChupaChups;
	(* the __NEW operator requires a stricktly typed pointer *)
	skittles			:POINTER TO SkittlesSour;
	(* the __NEW operator requires a stricktly typed pointer *)
	snickers			:POINTER TO SnickersBar;
	(* the __NEW operator requires a stricktly typed pointer *)
	twizzlers			:POINTER TO TwizzlersLicorizeTwists;
	(* the __NEW operator requires a stricktly typed pointer *)
	gobstopper			:POINTER TO WonkaGobstopper;
	(* return value is just a candy *)
	candy				:POINTER TO AbstractCandy;
END_VAR
getNewCandy REF= 0;
RETURN(THIS^.isCandyTypeInvalidForMachine(candyType));

CASE candyType OF
CandyTypes.CANDY_BARS,
CandyTypes.CARAMEL_CANDY,
CandyTypes.CHOCOLATE_CANDY:
	snickers := __NEW(SnickersBar());
	candy := snickers;
CandyTypes.CANDY_CORN,
CandyTypes.GUMMY_CANDY:
	candyCorn := __NEW(BrachsCandyCorn());
	candy := candyCorn;
CandyTypes.CANDY_STICKS:
	bobsStripes := __NEW(BobsSweetStripes());
	candy := bobsStripes;
CandyTypes.HARD_CANDY,
CandyTypes.LOLLIPOPS:
	chupChups := __NEW(ChupaChups());
	candy := chupChups;
CandyTypes.JAWBREAKERS:
	gobstopper := __NEW(WonkaGobstopper());
	candy := gobstopper;
CandyTypes.LICORICE_CANDY:
	twizzlers := __NEW(TwizzlersLicorizeTwists());
	candy := twizzlers;
CandyTypes.MINTS:
	altoids := __NEW(Altoids());
	candy := altoids;
CandyTypes.SOUR_CANDY:
	skittles := __NEW(SkittlesSour());
	candy := skittles;
ELSE
	RETURN;	
END_CASE

RETURN(candy <= 0);
getNewCandy REF= candy^;
END_METHOD

END_FUNCTION_BLOCK

// ---- Candies/Classes/Altoids.TcPOU
(*

short summary
=============
A specialized candy. It can be consumed by any candy consumer.
It supports dynamic creation. Furthermore, it calls the method 
AbstractCandy.initializeDispatchers after FB_init.

legal notes
===========
SPDX-FileCopyrightText: © 2024 ekvip automation GmbH <info@ekvip.de>
SPDX-License-Identifier: Apache-2.0
For details check: Apache-2.0_

.. _Apache-2.0: https://www.apache.org/licenses/LICENSE-2.0

*)

{attribute 'enable_dynamic_creation'}
{attribute 'call_after_init'}
FUNCTION_BLOCK FINAL Altoids EXTENDS AbstractCandy
VAR_INPUT
END_VAR
VAR_OUTPUT
END_VAR
VAR
END_VAR

(*

short summary
=============
it initializes the amount, the candy name and 
the binary coded candy type  

legal notes
===========
SPDX-FileCopyrightText: © 2024 ekvip automation GmbH <info@ekvip.de>
SPDX-License-Identifier: Apache-2.0
For details check: Apache-2.0_

.. _Apache-2.0: https://www.apache.org/licenses/LICENSE-2.0

*)

METHOD FB_init :BOOL
VAR_INPUT
	(* if TRUE, the retain variables are initialized (warm start / cold start) *)
	bInitRetains	:BOOL;
	(* if TRUE, the instance afterwards gets moved into the copy code (online change) *)
	bInCopyCode		:BOOL;
END_VAR
THIS^.amount := 50;
THIS^.name := 'Altoids Classic Peppermint';
THIS^.candyType := CandyTypes.MINTS;
END_METHOD

END_FUNCTION_BLOCK

// ---- Candies/Classes/BobsSweetStripes.TcPOU
(*

short summary
=============
A specialized candy. It can be consumed by any candy consumer.
It supports dynamic creation. Furthermore, it calls the method 
AbstractCandy.initializeDispatchers after FB_init.

legal notes
===========
SPDX-FileCopyrightText: © 2024 ekvip automation GmbH <info@ekvip.de>
SPDX-License-Identifier: Apache-2.0
For details check: Apache-2.0_

.. _Apache-2.0: https://www.apache.org/licenses/LICENSE-2.0

*)

{attribute 'enable_dynamic_creation'}
{attribute 'call_after_init'}
FUNCTION_BLOCK FINAL BobsSweetStripes EXTENDS AbstractCandy
VAR_INPUT
END_VAR
VAR_OUTPUT
END_VAR
VAR
END_VAR

(*

short summary
=============
it initializes the amount, the candy name and 
the binary coded candy type  

legal notes
===========
SPDX-FileCopyrightText: © 2024 ekvip automation GmbH <info@ekvip.de>
SPDX-License-Identifier: Apache-2.0
For details check: Apache-2.0_

.. _Apache-2.0: https://www.apache.org/licenses/LICENSE-2.0

*)

METHOD FB_init :BOOL
VAR_INPUT
	(* if TRUE, the retain variables are initialized (warm start / cold start) *)
	bInitRetains	:BOOL;
	(* if TRUE, the instance afterwards gets moved into the copy code (online change) *)
	bInCopyCode		:BOOL;
END_VAR
THIS^.amount := 282;
THIS^.name := 'Bobs Sweet Stripes';
THIS^.candyType := CandyTypes.CANDY_STICKS OR CandyTypes.MINTS OR CandyTypes.HARD_CANDY;
END_METHOD

END_FUNCTION_BLOCK

// ---- Candies/Classes/BrachsCandyCorn.TcPOU
(*

short summary
=============
A specialized candy. It can be consumed by any candy consumer.
It supports dynamic creation. Furthermore, it calls the method 
AbstractCandy.initializeDispatchers after FB_init.

legal notes
===========
SPDX-FileCopyrightText: © 2024 ekvip automation GmbH <info@ekvip.de>
SPDX-License-Identifier: Apache-2.0
For details check: Apache-2.0_

.. _Apache-2.0: https://www.apache.org/licenses/LICENSE-2.0

*)

{attribute 'enable_dynamic_creation'}
{attribute 'call_after_init'}
FUNCTION_BLOCK FINAL BrachsCandyCorn EXTENDS AbstractCandy
VAR_INPUT
END_VAR
VAR_OUTPUT
END_VAR
VAR
END_VAR

(*

short summary
=============
it initializes the amount, the candy name and 
the binary coded candy type  

legal notes
===========
SPDX-FileCopyrightText: © 2024 ekvip automation GmbH <info@ekvip.de>
SPDX-License-Identifier: Apache-2.0
For details check: Apache-2.0_

.. _Apache-2.0: https://www.apache.org/licenses/LICENSE-2.0

*)

METHOD FB_init :BOOL
VAR_INPUT
	(* if TRUE, the retain variables are initialized (warm start / cold start) *)
	bInitRetains	:BOOL;
	(* if TRUE, the instance afterwards gets moved into the copy code (online change) *)
	bInCopyCode		:BOOL;
END_VAR
THIS^.amount := 312;
THIS^.name := 'Brach$'s Candy Corn';
THIS^.candyType := CandyTypes.GUMMY_CANDY OR CandyTypes.CANDY_CORN;
END_METHOD

END_FUNCTION_BLOCK

// ---- Candies/Classes/ChupaChups.TcPOU
(*

short summary
=============
A specialized candy. It can be consumed by any candy consumer.
It supports dynamic creation. Furthermore, it calls the method 
AbstractCandy.initializeDispatchers after FB_init.

legal notes
===========
SPDX-FileCopyrightText: © 2024 ekvip automation GmbH <info@ekvip.de>
SPDX-License-Identifier: Apache-2.0
For details check: Apache-2.0_

.. _Apache-2.0: https://www.apache.org/licenses/LICENSE-2.0

*)

{attribute 'enable_dynamic_creation'}
{attribute 'call_after_init'}
FUNCTION_BLOCK FINAL ChupaChups EXTENDS AbstractCandy
VAR_INPUT
END_VAR
VAR_OUTPUT
END_VAR
VAR
END_VAR

(*

short summary
=============
it initializes the amount, the candy name and 
the binary coded candy type  

legal notes
===========
SPDX-FileCopyrightText: © 2024 ekvip automation GmbH <info@ekvip.de>
SPDX-License-Identifier: Apache-2.0
For details check: Apache-2.0_

.. _Apache-2.0: https://www.apache.org/licenses/LICENSE-2.0

*)

METHOD FB_init :BOOL
VAR_INPUT
	(* if TRUE, the retain variables are initialized (warm start / cold start) *)
	bInitRetains	:BOOL;
	(* if TRUE, the instance afterwards gets moved into the copy code (online change) *)
	bInCopyCode		:BOOL;
END_VAR
THIS^.amount := 120;
THIS^.name := 'Chupa Chups Sour';
THIS^.candyType := CandyTypes.LOLLIPOPS OR CandyTypes.SOUR_CANDY OR CandyTypes.HARD_CANDY;
END_METHOD

END_FUNCTION_BLOCK

// ---- Candies/Classes/SkittlesSour.TcPOU
(*

short summary
=============
A specialized candy. It can be consumed by any candy consumer.
It supports dynamic creation. Furthermore, it calls the method 
AbstractCandy.initializeDispatchers after FB_init.

legal notes
===========
SPDX-FileCopyrightText: © 2024 ekvip automation GmbH <info@ekvip.de>
SPDX-License-Identifier: Apache-2.0
For details check: Apache-2.0_

.. _Apache-2.0: https://www.apache.org/licenses/LICENSE-2.0

*)

{attribute 'enable_dynamic_creation'}
{attribute 'call_after_init'}
FUNCTION_BLOCK FINAL SkittlesSour EXTENDS AbstractCandy
VAR_INPUT
END_VAR
VAR_OUTPUT
END_VAR
VAR
END_VAR

(*

short summary
=============
it initializes the amount, the candy name and 
the binary coded candy type  

legal notes
===========
SPDX-FileCopyrightText: © 2024 ekvip automation GmbH <info@ekvip.de>
SPDX-License-Identifier: Apache-2.0
For details check: Apache-2.0_

.. _Apache-2.0: https://www.apache.org/licenses/LICENSE-2.0

*)

METHOD FB_init :BOOL
VAR_INPUT
	(* if TRUE, the retain variables are initialized (warm start / cold start) *)
	bInitRetains	:BOOL;
	(* if TRUE, the instance afterwards gets moved into the copy code (online change) *)
	bInCopyCode		:BOOL;
END_VAR
THIS^.amount := 160;
THIS^.name := 'Skittles Crazy Sours';
THIS^.candyType := CandyTypes.SOUR_CANDY;
END_METHOD

END_FUNCTION_BLOCK

// ---- Candies/Classes/SnickersBar.TcPOU
(*

short summary
=============
A specialized candy. It can be consumed by any candy consumer.
It supports dynamic creation. Furthermore, it calls the method 
AbstractCandy.initializeDispatchers after FB_init.

legal notes
===========
SPDX-FileCopyrightText: © 2024 ekvip automation GmbH <info@ekvip.de>
SPDX-License-Identifier: Apache-2.0
For details check: Apache-2.0_

.. _Apache-2.0: https://www.apache.org/licenses/LICENSE-2.0

*)

{attribute 'enable_dynamic_creation'}
{attribute 'call_after_init'}
FUNCTION_BLOCK FINAL SnickersBar EXTENDS AbstractCandy
VAR_INPUT
END_VAR
VAR_OUTPUT
END_VAR
VAR
END_VAR

(*

short summary
=============
it initializes the amount, the candy name and 
the binary coded candy type  

legal notes
===========
SPDX-FileCopyrightText: © 2024 ekvip automation GmbH <info@ekvip.de>
SPDX-License-Identifier: Apache-2.0
For details check: Apache-2.0_

.. _Apache-2.0: https://www.apache.org/licenses/LICENSE-2.0

*)

METHOD FB_init :BOOL
VAR_INPUT
	(* if TRUE, the retain variables are initialized (warm start / cold start) *)
	bInitRetains	:BOOL;
	(* if TRUE, the instance afterwards gets moved into the copy code (online change) *)
	bInCopyCode		:BOOL;
END_VAR
THIS^.amount := 51;
THIS^.name := 'Snickers';
THIS^.candyType := CandyTypes.CANDY_BARS OR CandyTypes.CHOCOLATE_CANDY OR CandyTypes.CARAMEL_CANDY;
END_METHOD

END_FUNCTION_BLOCK

// ---- Candies/Classes/TwizzlersLicorizeTwists.TcPOU
(*

short summary
=============
A specialized candy. It can be consumed by any candy consumer.
It supports dynamic creation. Furthermore, it calls the method 
AbstractCandy.initializeDispatchers after FB_init.

legal notes
===========
SPDX-FileCopyrightText: © 2024 ekvip automation GmbH <info@ekvip.de>
SPDX-License-Identifier: Apache-2.0
For details check: Apache-2.0_

.. _Apache-2.0: https://www.apache.org/licenses/LICENSE-2.0

*)

{attribute 'enable_dynamic_creation'}
{attribute 'call_after_init'}
FUNCTION_BLOCK FINAL TwizzlersLicorizeTwists EXTENDS AbstractCandy
VAR_INPUT
END_VAR
VAR_OUTPUT
END_VAR
VAR
END_VAR

(*

short summary
=============
it initializes the amount, the candy name and 
the binary coded candy type  

legal notes
===========
SPDX-FileCopyrightText: © 2024 ekvip automation GmbH <info@ekvip.de>
SPDX-License-Identifier: Apache-2.0
For details check: Apache-2.0_

.. _Apache-2.0: https://www.apache.org/licenses/LICENSE-2.0

*)

METHOD FB_init :BOOL
VAR_INPUT
	(* if TRUE, the retain variables are initialized (warm start / cold start) *)
	bInitRetains	:BOOL;
	(* if TRUE, the instance afterwards gets moved into the copy code (online change) *)
	bInCopyCode		:BOOL;
END_VAR
THIS^.amount := 454;
THIS^.name := 'Twizzlers Black Licorice Twists';
THIS^.candyType := CandyTypes.LICORICE_CANDY OR CandyTypes.GUMMY_CANDY;
END_METHOD

END_FUNCTION_BLOCK

// ---- Candies/Classes/WonkaGobstopper.TcPOU
(*

short summary
=============
A specialized candy. It can be consumed by any candy consumer.
It supports dynamic creation. Furthermore, it calls the method 
AbstractCandy.initializeDispatchers after FB_init.

legal notes
===========
SPDX-FileCopyrightText: © 2024 ekvip automation GmbH <info@ekvip.de>
SPDX-License-Identifier: Apache-2.0
For details check: Apache-2.0_

.. _Apache-2.0: https://www.apache.org/licenses/LICENSE-2.0

*)

{attribute 'enable_dynamic_creation'}
{attribute 'call_after_init'}
FUNCTION_BLOCK FINAL WonkaGobstopper EXTENDS AbstractCandy
VAR_INPUT
END_VAR
VAR_OUTPUT
END_VAR
VAR
END_VAR

(*

short summary
=============
it initializes the amount, the candy name and 
the binary coded candy type  

legal notes
===========
SPDX-FileCopyrightText: © 2024 ekvip automation GmbH <info@ekvip.de>
SPDX-License-Identifier: Apache-2.0
For details check: Apache-2.0_

.. _Apache-2.0: https://www.apache.org/licenses/LICENSE-2.0

*)

METHOD FB_init :BOOL
VAR_INPUT
	(* if TRUE, the retain variables are initialized (warm start / cold start) *)
	bInitRetains	:BOOL;
	(* if TRUE, the instance afterwards gets moved into the copy code (online change) *)
	bInCopyCode		:BOOL;
END_VAR
THIS^.amount := 141;
THIS^.name := 'Wonka Gobstopper';
THIS^.candyType := CandyTypes.JAWBREAKERS OR CandyTypes.SOUR_CANDY OR CandyTypes.HARD_CANDY;
END_METHOD

END_FUNCTION_BLOCK

// ---- CandyMachineProvider/Classes/NinjaIncCandyMachineProvider.TcPOU
(*

short summary
=============
here you'll find the best candy vending machines
on the market

legal notes
===========
SPDX-FileCopyrightText: © 2024 ekvip automation GmbH <info@ekvip.de>
SPDX-License-Identifier: Apache-2.0
For details check: Apache-2.0_

.. _Apache-2.0: https://www.apache.org/licenses/LICENSE-2.0

*)

FUNCTION_BLOCK NinjaIncCandyMachineProvider EXTENDS CandyMachineProvider
VAR_STAT
	(* the candy machine for greedy ninja monkeys *)
	greedyMachine	    :GreedyCandyMachine();
	(* the candy machine for picky ninja monkeys *) 
	pickyMachine		:PickyCandyMachine();
END_VAR

METHOD FB_Init :BOOL
VAR_INPUT
	(* TRUE: the retain variables are initialized (reset warm / reset cold) *)
    bInitRetains: BOOL;
	(* TRUE: the instance will be copied to the copy code afterward (online change) *)
    bInCopyCode: BOOL;
	(* Ninjas have a individual consume behavior and nina inc respects it *)
	consumerType :ConsumerTypes;
END_VAR
CASE consumerType OF
ConsumerTypes.GREEDY:
	customCandyMachine REF= THIS^.greedyMachine;	
ConsumerTypes.PICKY:
	customCandyMachine REF= THIS^.pickyMachine;
ELSE;// just use the default candy machine
END_CASE
END_METHOD

END_FUNCTION_BLOCK

// ---- CandyMachine/Classes/GreedyCandyMachine.TcPOU
(*

short summary
=============
A candy vending machine for the greedy eaters.
It tries to provide candies with a high amount. 

legal notes
===========
SPDX-FileCopyrightText: © 2024 ekvip automation GmbH <info@ekvip.de>
SPDX-License-Identifier: Apache-2.0
For details check: Apache-2.0_

.. _Apache-2.0: https://www.apache.org/licenses/LICENSE-2.0

*)

FUNCTION_BLOCK FINAL GreedyCandyMachine EXTENDS AbstractCandyMachine

(*

short summary
=============
want some, get some
this method provides the candies

legal notes
===========
SPDX-FileCopyrightText: © 2024 ekvip automation GmbH <info@ekvip.de>
SPDX-License-Identifier: Apache-2.0
For details check: Apache-2.0_

.. _Apache-2.0: https://www.apache.org/licenses/LICENSE-2.0

*)

METHOD  getNewCandy :REFERENCE TO AbstractCandy
VAR_INPUT
	(*preferred candy type, it must be a pure candy type *)
	candyType	:CandyTypes;
END_VAR
VAR
	(* the __NEW operator requires a stricktly typed pointer *)
	alpenliebe			:POINTER TO Alpenliebe;
	(* the __NEW operator requires a stricktly typed pointer *)
	bobsStripes			:POINTER TO BobsSweetStripes;
	(* the __NEW operator requires a stricktly typed pointer *)
	candyCorn			:POINTER TO BrachsCandyCorn;
	(* the __NEW operator requires a stricktly typed pointer *)
	chupChups			:POINTER TO ChupaChups;
	(* the __NEW operator requires a stricktly typed pointer *)
	skittles			:POINTER TO SkittlesSour;
	(* the __NEW operator requires a stricktly typed pointer *)
	snickers			:POINTER TO SnickersBar;
	(* the __NEW operator requires a stricktly typed pointer *)
	twizzlers			:POINTER TO TwizzlersLicorizeTwists;
	(* the __NEW operator requires a stricktly typed pointer *)
	gobstopper			:POINTER TO WonkaGobstopper;
	(* return value is just a candy *)
	candy				:POINTER TO AbstractCandy;
END_VAR
getNewCandy REF= 0;
RETURN(THIS^.isCandyTypeInvalidForMachine(candyType));

CASE candyType OF
CandyTypes.CANDY_BARS,
CandyTypes.CHOCOLATE_CANDY:
	snickers := __NEW(SnickersBar());
	candy := snickers;
CandyTypes.CANDY_CORN:
	candyCorn := __NEW(BrachsCandyCorn());
	candy := candyCorn;
CandyTypes.CANDY_STICKS,
CandyTypes.MINTS,
CandyTypes.HARD_CANDY:
	bobsStripes := __NEW(BobsSweetStripes());
	candy := bobsStripes;
CandyTypes.CARAMEL_CANDY:
	alpenliebe := __NEW(Alpenliebe());
	candy := alpenliebe;
CandyTypes.GUMMY_CANDY,
CandyTypes.LICORICE_CANDY:
	twizzlers := __NEW(TwizzlersLicorizeTwists());
	candy := twizzlers;
CandyTypes.JAWBREAKERS:
	gobstopper := __NEW(WonkaGobstopper());
	candy := gobstopper;
CandyTypes.LOLLIPOPS:;
	chupChups := __NEW(ChupaChups());
	candy := chupChups;
CandyTypes.SOUR_CANDY:;
	skittles := __NEW(SkittlesSour());
	candy := skittles;
ELSE
	RETURN;
END_CASE

RETURN(candy <= 0);
getNewCandy REF= candy^;
END_METHOD

END_FUNCTION_BLOCK

// ---- Candies/Classes/Alpenliebe.TcPOU
(*

short summary
=============
A specialized candy. It can be consumed by any candy consumer.
It supports dynamic creation. Furthermore, it calls the method 
AbstractCandy.initializeDispatchers after FB_init.

legal notes
===========
SPDX-FileCopyrightText: © 2024 ekvip automation GmbH <info@ekvip.de>
SPDX-License-Identifier: Apache-2.0
For details check: Apache-2.0_

.. _Apache-2.0: https://www.apache.org/licenses/LICENSE-2.0

*)

{attribute 'enable_dynamic_creation'}
{attribute 'call_after_init'}
FUNCTION_BLOCK FINAL Alpenliebe EXTENDS AbstractCandy
VAR_INPUT
END_VAR
VAR_OUTPUT
END_VAR
VAR
END_VAR

(*

short summary
=============
it initializes the amount, the candy name and 
the binary coded candy type  

legal notes
===========
SPDX-FileCopyrightText: © 2024 ekvip automation GmbH <info@ekvip.de>
SPDX-License-Identifier: Apache-2.0
For details check: Apache-2.0_

.. _Apache-2.0: https://www.apache.org/licenses/LICENSE-2.0

*)

METHOD FB_init :BOOL
VAR_INPUT
	(* if TRUE, the retain variables are initialized (warm start / cold start) *)
	bInitRetains	:BOOL;
	(* if TRUE, the instance afterwards gets moved into the copy code (online change) *)
	bInCopyCode		:BOOL;
END_VAR
THIS^.amount := 156;
THIS^.name := 'Alpenliebe Gold';
THIS^.candyType := CandyTypes.HARD_CANDY OR CandyTypes.CARAMEL_CANDY;
END_METHOD

END_FUNCTION_BLOCK

// ---- CandyMachine/Classes/PickyCandyMachine.TcPOU
(*

short summary
=============
a candy vending machine for the picky eaters. 
It tries to provide candies that match the desired candy type. 

legal notes
===========
SPDX-FileCopyrightText: © 2024 ekvip automation GmbH <info@ekvip.de>
SPDX-License-Identifier: Apache-2.0
For details check: Apache-2.0_

.. _Apache-2.0: https://www.apache.org/licenses/LICENSE-2.0

*)

FUNCTION_BLOCK FINAL PickyCandyMachine EXTENDS AbstractCandyMachine

(*

short summary
=============
want some, get some
this method provides the candies

legal notes
===========
SPDX-FileCopyrightText: © 2024 ekvip automation GmbH <info@ekvip.de>
SPDX-License-Identifier: Apache-2.0
For details check: Apache-2.0_

.. _Apache-2.0: https://www.apache.org/licenses/LICENSE-2.0

*)

